  [805] = {x=8.913773, y=-27.596676, z=96.640035, rx=178.000889, ry=-0.000182, rz=-0.000291, shoulder=lefty, elbow=epositive, wrist=wpositive, fatherId=frmaster[2]}
  [806] = {x=7.923867, y=-27.612388, z=96.649585, rx=177.998895, ry=0.000218, rz=-0.000016, shoulder=lefty, elbow=epositive, wrist=wpositive, fatherId=frmaster[2]}
  [807] = {x=6.93352, y=-27.623246, z=96.64007, rx=178.000793, ry=-0.000277, rz=-0.000734, shoulder=lefty, elbow=epositive, wrist=wpositive, fatherId=frmaster[2]}
  [808] = {x=5.944819, y=-27.63732, z=96.640862, rx=178.000734, ry=-0.000326, rz=-0.000446, shoulder=lefty, elbow=epositive, wrist=wpositive, fatherId=frmaster[2]}
  [809] = {x=4.947952, y=-27.654261, z=96.646832, rx=177.999684, ry=-0.000194, rz=-0.000153, shoulder=lefty, elbow=epositive, wrist=wpositive, fatherId=frmaster[2]}
  [810] = {x=3.960147, y=-27.66522, z=96.643162, rx=178.000587, ry=-0.000463, rz=0.000148, shoulder=lefty, elbow=epositive, wrist=wpositive, fatherId=frmaster[2]}
  [811] = {x=2.973867, y=-27.679396, z=96.640369, rx=178.000507, ry=-0.000514, rz=-0.000545, shoulder=lefty, elbow=epositive, wrist=wpositive, fatherId=frmaster[2]}
  [812] = {x=1.979877, y=-27.693391, z=96.637557, rx=178.000612, ry=0.000317, rz=0.000105, shoulder=lefty, elbow=epositive, wrist=wpositive, fatherId=frmaster[2]}
  [813] = {x=0.995231, y=-27.707402, z=96.644933, rx=177.999539, ry=0.000476, rz=-0.000577, shoulder=lefty, elbow=epositive, wrist=wpositive, fatherId=frmaster[2]}
  [814] = {x=0.001401, y=-27.720204, z=96.642841, rx=178.000405, ry=0.000175, rz=-0.000253, shoulder=lefty, elbow=epositive, wrist=wpositive, fatherId=frmaster[2]}
  [815] = {x=-0.983292, y=-27.726863, z=96.644847, rx=178.000296, ry=0.00012, rz=0.000079, shoulder=lefty, elbow=epositive, wrist=wpositive, fatherId=frmaster[2]}
  [816] = {x=-1.976258, y=-27.736283, z=96.642626, rx=178.00017, ry=0.000028, rz=-0.000584, shoulder=lefty, elbow=epositive, wrist=wpositive, fatherId=frmaster[2]}
  [817] = {x=-2.968913, y=-27.743412, z=96.64032, rx=178.000038, ry=-0.000065, rz=-0.000241, shoulder=lefty, elbow=epositive, wrist=wpositive, fatherId=frmaster[2]}
  [818] = {x=-3.960489, y=-27.75152, z=96.648216, rx=177.999898, ry=-0.000158, rz=0.000105, shoulder=lefty, elbow=epositive, wrist=wpositive, fatherId=frmaster[2]}
  [819] = {x=-4.9516, y=-27.758484, z=96.646675, rx=177.999752, ry=-0.000253, rz=0.000459, shoulder=lefty, elbow=epositive, wrist=wpositive, fatherId=frmaster[2]}
  [820] = {x=-5.941493, y=-27.767594, z=96.645991, rx=177.999599, ry=-0.000348, rz=-0.000182, shoulder=lefty, elbow=epositive, wrist=wpositive, fatherId=frmaster[2]}
  [821] = {x=-6.929953, y=-27.77423, z=96.645219, rx=177.999623, ry=0.000476, rz=0.000527, shoulder=lefty, elbow=epositive, wrist=wpositive, fatherId=frmaster[2]}
  [822] = {x=-7.918944, y=-27.78043, z=96.640137, rx=178.000435, ry=0.000184, rz=-0.000102, shoulder=lefty, elbow=epositive, wrist=wpositive, fatherId=frmaster[2]}
  [823] = {x=-8.907014, y=-27.787247, z=96.64016, rx=178.000259, ry=0.000088, rz=0.000274, shoulder=lefty, elbow=epositive, wrist=wpositive, fatherId=frmaster[2]}
  [824] = {x=-9.894404, y=-27.7935, z=96.645241, rx=178.000077, ry=-0.000009, rz=-0.000346, shoulder=lefty, elbow=epositive, wrist=wpositive, fatherId=frmaster[2]}
  [825] = {x=-10.890105, y=-27.802454, z=96.646129, rx=177.999879, ry=-0.000143, rz=0.000038, shoulder=lefty, elbow=epositive, wrist=wpositive, fatherId=frmaster[2]}
  [826] = {x=-11.875867, y=-27.809861, z=96.64268, rx=177.999682, ry=-0.000242, rz=-0.000571, shoulder=lefty, elbow=epositive, wrist=wpositive, fatherId=frmaster[2]}
  [827] = {x=-12.870091, y=-27.818836, z=96.644369, rx=177.99947, ry=-0.000378, rz=-0.000177, shoulder=lefty, elbow=epositive, wrist=wpositive, fatherId=frmaster[2]}
  [828] = {x=-13.853395, y=-27.824988, z=96.651034, rx=177.999433, ry=0.000443, rz=-0.000429, shoulder=lefty, elbow=epositive, wrist=wpositive, fatherId=frmaster[2]}
  [829] = {x=-14.846607, y=-27.832289, z=96.639048, rx=178.000188, ry=0.000122, rz=-0.000021, shoulder=lefty, elbow=epositive, wrist=wpositive, fatherId=frmaster[2]}
  [830] = {x=-15.838709, y=-27.840827, z=96.646606, rx=177.999955, ry=-0.000014, rz=0.000386, shoulder=lefty, elbow=epositive, wrist=wpositive, fatherId=frmaster[2]}
  [831] = {x=-16.830382, y=-27.848304, z=96.64479, rx=177.999714, ry=-0.000152, rz=-0.0002, shoulder=lefty, elbow=epositive, wrist=wpositive, fatherId=frmaster[2]}
  [832] = {x=-17.821399, y=-27.855287, z=96.648035, rx=177.999466, ry=-0.00029, rz=0.000218, shoulder=lefty, elbow=epositive, wrist=wpositive, fatherId=frmaster[2]}
  [833] = {x=-18.810516, y=-27.862721, z=96.647037, rx=177.999375, ry=0.000492, rz=0.000994, shoulder=lefty, elbow=epositive, wrist=wpositive, fatherId=frmaster[2]}
  [834] = {x=-19.800203, y=-27.869818, z=96.641773, rx=178.000097, ry=0.000178, rz=0.000423, shoulder=lefty, elbow=epositive, wrist=wpositive, fatherId=frmaster[2]}
  [835] = {x=-20.789037, y=-27.877666, z=96.641616, rx=177.999827, ry=0.000038, rz=-0.000146, shoulder=lefty, elbow=epositive, wrist=wpositive, fatherId=frmaster[2]}
  [836] = {x=-21.777233, y=-27.885073, z=96.64652, rx=177.999551, ry=-0.000102, rz=0.000288, shoulder=lefty, elbow=epositive, wrist=wpositive, fatherId=frmaster[2]}
  [837] = {x=-22.765223, y=-27.890266, z=96.642039, rx=178.000254, ry=-0.000411, rz=-0.00027, shoulder=lefty, elbow=epositive, wrist=wpositive, fatherId=frmaster[2]}
  [838] = {x=-23.75984, y=-27.900874, z=96.647894, rx=177.999124, ry=0.0005, rz=0.000527, shoulder=lefty, elbow=epositive, wrist=wpositive, fatherId=frmaster[2]}
  [839] = {x=-24.746454, y=-27.906358, z=96.644261, rx=177.999812, ry=0.000193, rz=-0.000023, shoulder=lefty, elbow=epositive, wrist=wpositive, fatherId=frmaster[2]}
  [840] = {x=-25.741373, y=-27.914513, z=96.645809, rx=177.999498, ry=0.000015, rz=0.000428, shoulder=lefty, elbow=epositive, wrist=wpositive, fatherId=frmaster[2]}
  [841] = {x=-26.726631, y=-27.920333, z=96.643032, rx=178.000174, ry=-0.000289, rz=-0.000115, shoulder=lefty, elbow=epositive, wrist=wpositive, fatherId=frmaster[2]}
  [842] = {x=-27.719082, y=-27.928635, z=96.64543, rx=177.999995, ry=0.000455, rz=0.000701, shoulder=lefty, elbow=epositive, wrist=wpositive, fatherId=frmaster[2]}
  [843] = {x=-28.702817, y=-27.936049, z=96.643558, rx=177.999668, ry=0.000311, rz=-0.000835, shoulder=lefty, elbow=epositive, wrist=wpositive, fatherId=frmaster[2]}
  [844] = {x=-29.695588, y=-27.941964, z=96.64167, rx=178.000314, ry=-0.000024, rz=-0.000367, shoulder=lefty, elbow=epositive, wrist=wpositive, fatherId=frmaster[2]}
  [845] = {x=-30.687149, y=-27.951588, z=96.640743, rx=177.999965, ry=-0.000203, rz=0.000102, shoulder=lefty, elbow=epositive, wrist=wpositive, fatherId=frmaster[2]}
  [846] = {x=-31.678617, y=-27.957901, z=96.639728, rx=178.000598, ry=-0.000535, rz=-0.000423, shoulder=lefty, elbow=epositive, wrist=wpositive, fatherId=frmaster[2]}
  [847] = {x=-32.668177, y=-27.964899, z=96.643809, rx=178.000376, ry=0.000208, rz=0.000413, shoulder=lefty, elbow=epositive, wrist=wpositive, fatherId=frmaster[2]}
  [848] = {x=-33.658182, y=-27.972864, z=96.643712, rx=178.000006, ry=0.000028, rz=-0.000106, shoulder=lefty, elbow=epositive, wrist=wpositive, fatherId=frmaster[2]}
  [849] = {x=-34.647604, y=-27.980501, z=96.648675, rx=177.999629, ry=-0.000153, rz=0.000375, shoulder=lefty, elbow=epositive, wrist=wpositive, fatherId=frmaster[2]}
  [850] = {x=-35.636361, y=-27.988956, z=96.64946, rx=177.999245, ry=-0.000335, rz=-0.000139, shoulder=lefty, elbow=epositive, wrist=wpositive, fatherId=frmaster[2]}
  [851] = {x=-36.623808, y=-27.995104, z=96.640917, rx=177.999977, ry=0.000261, rz=-0.000282, shoulder=lefty, elbow=epositive, wrist=wpositive, fatherId=frmaster[2]}
  [852] = {x=-37.620853, y=-28.002846, z=96.646798, rx=177.99957, ry=0.000043, rz=0.000209, shoulder=lefty, elbow=epositive, wrist=wpositive, fatherId=frmaster[2]}
  [853] = {x=-38.608373, y=-28.008476, z=96.639117, rx=178.001145, ry=-0.000417, rz=-0.000292, shoulder=lefty, elbow=epositive, wrist=wpositive, fatherId=frmaster[2]}
  [854] = {x=-39.593779, y=-28.016167, z=96.64585, rx=177.99987, ry=0.000462, rz=-0.000431, shoulder=lefty, elbow=epositive, wrist=wpositive, fatherId=frmaster[2]}
  [855] = {x=-40.58907, y=-28.025203, z=96.639191, rx=178.000432, ry=0.000108, rz=0.000072, shoulder=lefty, elbow=epositive, wrist=wpositive, fatherId=frmaster[2]}
  [856] = {x=-41.574591, y=-28.032435, z=96.646785, rx=178.000006, ry=-0.000073, rz=-0.000427, shoulder=lefty, elbow=epositive, wrist=wpositive, fatherId=frmaster[2]}
  [857] = {x=-42.568912, y=-28.040341, z=96.645196, rx=177.999564, ry=-0.000293, rz=0.000081, shoulder=lefty, elbow=epositive, wrist=wpositive, fatherId=frmaster[2]}
  [858] = {x=-43.552519, y=-28.046198, z=96.63933, rx=178.000236, ry=0.000315, rz=-0.000039, shoulder=lefty, elbow=epositive, wrist=wpositive, fatherId=frmaster[2]}
  [859] = {x=-44.545849, y=-28.053507, z=96.638612, rx=178.000771, ry=-0.000031, rz=-0.000527, shoulder=lefty, elbow=epositive, wrist=wpositive, fatherId=frmaster[2]}
  [860] = {x=-45.538493, y=-28.061772, z=96.642998, rx=178.000309, ry=-0.000249, rz=-0.000015, shoulder=lefty, elbow=epositive, wrist=wpositive, fatherId=frmaster[2]}
  [861] = {x=-46.529424, y=-28.070788, z=96.643232, rx=177.999953, ry=0.000454, rz=0.00087, shoulder=lefty, elbow=epositive, wrist=wpositive, fatherId=frmaster[2]}
  [862] = {x=-47.512248, y=-28.075214, z=96.643319, rx=178.000477, ry=0.000148, rz=-0.00061, shoulder=lefty, elbow=epositive, wrist=wpositive, fatherId=frmaster[2]}
  [863] = {x=-48.503627, y=-28.082047, z=96.639343, rx=178.000985, ry=-0.000191, rz=-0.000086, shoulder=lefty, elbow=epositive, wrist=wpositive, fatherId=frmaster[2]}
  [864] = {x=-49.494351, y=-28.08987, z=96.640474, rx=178.000495, ry=-0.00041, rz=-0.000563, shoulder=lefty, elbow=epositive, wrist=wpositive, fatherId=frmaster[2]}
  [865] = {x=-50.483444, y=-28.097352, z=96.646661, rx=178.000105, ry=0.000294, rz=-0.00067, shoulder=lefty, elbow=epositive, wrist=wpositive, fatherId=frmaster[2]}
  [866] = {x=-51.473202, y=-28.105824, z=96.639482, rx=178.000593, ry=-0.000041, rz=-0.000139, shoulder=lefty, elbow=epositive, wrist=wpositive, fatherId=frmaster[2]}
  [867] = {x=-52.471771, y=-28.113763, z=96.641589, rx=178.000072, ry=-0.000297, rz=0.00039, shoulder=lefty, elbow=epositive, wrist=wpositive, fatherId=frmaster[2]}
  [868] = {x=-53.459292, y=-28.122929, z=96.644577, rx=177.999656, ry=0.000406, rz=0.00029, shoulder=lefty, elbow=epositive, wrist=wpositive, fatherId=frmaster[2]}
  [869] = {x=-54.447712, y=-28.130227, z=96.647541, rx=177.999129, ry=0.000185, rz=-0.000177, shoulder=lefty, elbow=epositive, wrist=wpositive, fatherId=frmaster[2]}
  [870] = {x=-55.435743, y=-28.137278, z=96.646339, rx=177.99959, ry=-0.000144, rz=-0.000641, shoulder=lefty, elbow=epositive, wrist=wpositive, fatherId=frmaster[2]}
  [871] = {x=-56.422416, y=-28.142223, z=96.645109, rx=178.000141, ry=0.000452, rz=-0.000729, shoulder=lefty, elbow=epositive, wrist=wpositive, fatherId=frmaster[2]}
  [872] = {x=-57.41848, y=-28.152621, z=96.644972, rx=177.999584, ry=0.000195, rz=-0.000192, shoulder=lefty, elbow=epositive, wrist=wpositive, fatherId=frmaster[2]}
  [873] = {x=-58.405313, y=-28.158501, z=96.644693, rx=178.000025, ry=-0.000127, rz=-0.000651, shoulder=lefty, elbow=epositive, wrist=wpositive, fatherId=frmaster[2]}
  [874] = {x=-59.400791, y=-28.166654, z=96.640378, rx=178.00045, ry=-0.000484, rz=-0.000107, shoulder=lefty, elbow=epositive, wrist=wpositive, fatherId=frmaster[2]}
  [875] = {x=-60.385354, y=-28.174566, z=96.650304, rx=177.998977, ry=0.000318, rz=-0.000195, shoulder=lefty, elbow=epositive, wrist=wpositive, fatherId=frmaster[2]}
  [876] = {x=-61.380256, y=-28.180496, z=96.641817, rx=178.000384, ry=-0.000133, rz=0.000355, shoulder=lefty, elbow=epositive, wrist=wpositive, fatherId=frmaster[2]}
  [877] = {x=-62.365132, y=-28.18932, z=96.643487, rx=177.999802, ry=-0.000352, rz=-0.000101, shoulder=lefty, elbow=epositive, wrist=wpositive, fatherId=frmaster[2]}
  [878] = {x=-63.357812, y=-28.197297, z=96.64521, rx=177.999289, ry=0.000314, rz=-0.00018, shoulder=lefty, elbow=epositive, wrist=wpositive, fatherId=frmaster[2]}
  [879] = {x=-64.342146, y=-28.203971, z=96.642714, rx=177.999688, ry=0.000002, rz=-0.00063, shoulder=lefty, elbow=epositive, wrist=wpositive, fatherId=frmaster[2]}
  [880] = {x=-65.335411, y=-28.209874, z=96.640279, rx=178.000073, ry=-0.000344, rz=-0.000077, shoulder=lefty, elbow=epositive, wrist=wpositive, fatherId=frmaster[2]}
  [881] = {x=-66.326818, y=-28.218619, z=96.648026, rx=177.999534, ry=0.000325, rz=-0.000157, shoulder=lefty, elbow=epositive, wrist=wpositive, fatherId=frmaster[2]}
  [882] = {x=-67.319242, y=-28.225415, z=96.646555, rx=177.999904, ry=-0.000016, rz=0.000396, shoulder=lefty, elbow=epositive, wrist=wpositive, fatherId=frmaster[2]}
  [883] = {x=-66.317022, y=-28.225289, z=96.64487, rx=177.999542, ry=0.000364, rz=-0.000161, shoulder=lefty, elbow=epositive, wrist=wpositive, fatherId=frmaster[2]}
  [884] = {x=-65.324629, y=-28.226264, z=96.648325, rx=177.999086, ry=-0.000212, rz=-0.000098, shoulder=lefty, elbow=epositive, wrist=wpositive, fatherId=frmaster[2]}
  [885] = {x=-64.321617, y=-28.225732, z=96.647556, rx=177.999707, ry=0.000085, rz=-0.000655, shoulder=lefty, elbow=epositive, wrist=wpositive, fatherId=frmaster[2]}
  [886] = {x=-63.3274, y=-28.225595, z=96.646886, rx=177.999316, ry=0.000435, rz=-0.000209, shoulder=lefty, elbow=epositive, wrist=wpositive, fatherId=frmaster[2]}
  [887] = {x=-62.33406, y=-28.224115, z=96.642027, rx=178.000825, ry=-0.000322, rz=-0.000135, shoulder=lefty, elbow=epositive, wrist=wpositive, fatherId=frmaster[2]}
  [888] = {x=-61.329773, y=-28.223559, z=96.642231, rx=178.000429, ry=0.000066, rz=-0.000688, shoulder=lefty, elbow=epositive, wrist=wpositive, fatherId=frmaster[2]}
  [889] = {x=-60.334157, y=-28.224056, z=96.647574, rx=178.000018, ry=0.000422, rz=-0.000242, shoulder=lefty, elbow=epositive, wrist=wpositive, fatherId=frmaster[2]}
  [890] = {x=-59.339162, y=-28.225622, z=96.648809, rx=177.99951, ry=-0.000143, rz=-0.000168, shoulder=lefty, elbow=epositive, wrist=wpositive, fatherId=frmaster[2]}
  [891] = {x=-58.34288, y=-28.224981, z=96.640795, rx=178.000079, ry=0.000115, rz=0.000289, shoulder=lefty, elbow=epositive, wrist=wpositive, fatherId=frmaster[2]}
  [892] = {x=-57.345756, y=-28.227191, z=96.642969, rx=177.999648, ry=0.000477, rz=0.00074, shoulder=lefty, elbow=epositive, wrist=wpositive, fatherId=frmaster[2]}
  [893] = {x=-56.349631, y=-28.226272, z=96.645077, rx=178.000108, ry=-0.000186, rz=-0.000178, shoulder=lefty, elbow=epositive, wrist=wpositive, fatherId=frmaster[2]}
  [894] = {x=-55.352089, y=-28.224342, z=96.637971, rx=178.000657, ry=0.00007, rz=0.000284, shoulder=lefty, elbow=epositive, wrist=wpositive, fatherId=frmaster[2]}
  [895] = {x=-54.353676, y=-28.225231, z=96.641054, rx=178.000205, ry=0.000437, rz=0.000741, shoulder=lefty, elbow=epositive, wrist=wpositive, fatherId=frmaster[2]}
  [896] = {x=-53.355882, y=-28.226014, z=96.649205, rx=177.999645, ry=-0.000116, rz=-0.000174, shoulder=lefty, elbow=epositive, wrist=wpositive, fatherId=frmaster[2]}
  [897] = {x=-52.35665, y=-28.225759, z=96.648132, rx=177.999178, ry=0.000254, rz=0.00029, shoulder=lefty, elbow=epositive, wrist=wpositive, fatherId=frmaster[2]}
  [898] = {x=-51.357127, y=-28.22397, z=96.64284, rx=178.000693, ry=0.0004, rz=-0.000242, shoulder=lefty, elbow=epositive, wrist=wpositive, fatherId=frmaster[2]}
  [899] = {x=-50.367069, y=-28.22592, z=96.642773, rx=178.000098, ry=-0.000187, rz=0.000855, shoulder=lefty, elbow=epositive, wrist=wpositive, fatherId=frmaster[2]}
  [900] = {x=-49.366217, y=-28.226061, z=96.647685, rx=177.999611, ry=0.00019, rz=0.000322, shoulder=lefty, elbow=epositive, wrist=wpositive, fatherId=frmaster[2]}
  [901] = {x=-48.365182, y=-28.224052, z=96.64332, rx=178.000111, ry=0.000447, rz=-0.000203, shoulder=lefty, elbow=epositive, wrist=wpositive, fatherId=frmaster[2]}
  [902] = {x=-47.373462, y=-28.226399, z=96.649234, rx=177.999491, ry=-0.000132, rz=-0.000102, shoulder=lefty, elbow=epositive, wrist=wpositive, fatherId=frmaster[2]}
  [903] = {x=-46.371288, y=-28.224977, z=96.645782, rx=177.999976, ry=0.000126, rz=-0.000623, shoulder=lefty, elbow=epositive, wrist=wpositive, fatherId=frmaster[2]}
  [904] = {x=-45.377551, y=-28.22599, z=96.647509, rx=177.999453, ry=0.000472, rz=0.000855, shoulder=lefty, elbow=epositive, wrist=wpositive, fatherId=frmaster[2]}
  [905] = {x=-44.375338, y=-28.225258, z=96.644969, rx=177.999807, ry=-0.000192, rz=-0.000029, shoulder=lefty, elbow=epositive, wrist=wpositive, fatherId=frmaster[2]}
  [906] = {x=-43.380854, y=-28.223836, z=96.642461, rx=178.000262, ry=0.000028, rz=-0.000542, shoulder=lefty, elbow=epositive, wrist=wpositive, fatherId=frmaster[2]}
  [907] = {x=-42.385459, y=-28.225042, z=96.640892, rx=178.000711, ry=0.000248, rz=-0.000055, shoulder=lefty, elbow=epositive, wrist=wpositive, fatherId=frmaster[2]}
  [908] = {x=-41.390904, y=-28.224314, z=96.639287, rx=178.001029, ry=-0.000457, rz=0.00007, shoulder=lefty, elbow=epositive, wrist=wpositive, fatherId=frmaster[2]}
  [909] = {x=-40.394487, y=-28.224336, z=96.64278, rx=178.000471, ry=-0.000104, rz=0.000562, shoulder=lefty, elbow=epositive, wrist=wpositive, fatherId=frmaster[2]}
  [910] = {x=-39.388444, y=-28.222336, z=96.641987, rx=178.000907, ry=0.000151, rz=0.000059, shoulder=lefty, elbow=epositive, wrist=wpositive, fatherId=frmaster[2]}
  [911] = {x=-38.391912, y=-28.222977, z=96.64638, rx=178.000208, ry=-0.000415, rz=-0.000808, shoulder=lefty, elbow=epositive, wrist=wpositive, fatherId=frmaster[2]}
  [912] = {x=-37.402718, y=-28.225912, z=96.646671, rx=177.999621, ry=-0.000093, rz=0.000693, shoulder=lefty, elbow=epositive, wrist=wpositive, fatherId=frmaster[2]}
  [913] = {x=-36.403877, y=-28.226772, z=96.642665, rx=178.000027, ry=0.000126, rz=0.000199, shoulder=lefty, elbow=epositive, wrist=wpositive, fatherId=frmaster[2]}
  [914] = {x=-35.404647, y=-28.22558, z=96.647894, rx=177.999437, ry=0.000489, rz=0.000706, shoulder=lefty, elbow=epositive, wrist=wpositive, fatherId=frmaster[2]}
  [915] = {x=-34.406123, y=-28.224032, z=96.639617, rx=178.000682, ry=-0.000361, rz=-0.00014, shoulder=lefty, elbow=epositive, wrist=wpositive, fatherId=frmaster[2]}
  [916] = {x=-33.405599, y=-28.223217, z=96.645724, rx=178.000077, ry=0.000003, rz=-0.000627, shoulder=lefty, elbow=epositive, wrist=wpositive, fatherId=frmaster[2]}
  [917] = {x=-32.413596, y=-28.224812, z=96.638426, rx=178.000446, ry=0.000183, rz=-0.000106, shoulder=lefty, elbow=epositive, wrist=wpositive, fatherId=frmaster[2]}
  [918] = {x=-31.412876, y=-28.224513, z=96.645411, rx=177.999687, ry=-0.000371, rz=0.000054, shoulder=lefty, elbow=epositive, wrist=wpositive, fatherId=frmaster[2]}
  [919] = {x=-30.419445, y=-28.226537, z=96.648273, rx=177.999053, ry=-0.000037, rz=0.000578, shoulder=lefty, elbow=epositive, wrist=wpositive, fatherId=frmaster[2]}
  [920] = {x=-29.416847, y=-28.223345, z=96.64166, rx=178.000396, ry=0.000025, rz=0.000111, shoulder=lefty, elbow=epositive, wrist=wpositive, fatherId=frmaster[2]}
  [921] = {x=-28.422057, y=-28.225676, z=96.64538, rx=177.999749, ry=0.000361, rz=-0.000358, shoulder=lefty, elbow=epositive, wrist=wpositive, fatherId=frmaster[2]}
  [922] = {x=-27.428363, y=-28.224754, z=96.639699, rx=178.000922, ry=-0.000541, rz=-0.000177, shoulder=lefty, elbow=epositive, wrist=wpositive, fatherId=frmaster[2]}
  [923] = {x=-26.432518, y=-28.225634, z=96.639153, rx=178.00026, ry=-0.000204, rz=0.000364, shoulder=lefty, elbow=epositive, wrist=wpositive, fatherId=frmaster[2]}
  [924] = {x=-25.42709, y=-28.222996, z=96.643548, rx=178.000587, ry=0.00001, rz=-0.000091, shoulder=lefty, elbow=epositive, wrist=wpositive, fatherId=frmaster[2]}
  [925] = {x=-24.429846, y=-28.22409, z=96.643847, rx=177.999912, ry=0.000351, rz=-0.000542, shoulder=lefty, elbow=epositive, wrist=wpositive, fatherId=frmaster[2]}
  [926] = {x=-23.433165, y=-28.224831, z=96.639887, rx=178.000062, ry=-0.000394, rz=-0.000344, shoulder=lefty, elbow=epositive, wrist=wpositive, fatherId=frmaster[2]}
  [927] = {x=-22.434701, y=-28.224901, z=96.640978, rx=178.000359, ry=-0.000218, rz=-0.000787, shoulder=lefty, elbow=epositive, wrist=wpositive, fatherId=frmaster[2]}
  [928] = {x=-21.445055, y=-28.224708, z=96.642082, rx=178.00064, ry=-0.000079, rz=0.000775, shoulder=lefty, elbow=epositive, wrist=wpositive, fatherId=frmaster[2]}
  [929] = {x=-20.444948, y=-28.226127, z=96.644044, rx=177.999938, ry=0.000268, rz=0.00034, shoulder=lefty, elbow=epositive, wrist=wpositive, fatherId=frmaster[2]}
  [930] = {x=-19.444725, y=-28.224121, z=96.645899, rx=178.000215, ry=0.000443, rz=-0.00009, shoulder=lefty, elbow=epositive, wrist=wpositive, fatherId=frmaster[2]}
  [931] = {x=-18.453978, y=-28.224908, z=96.643598, rx=178.000312, ry=-0.000341, rz=0.000134, shoulder=lefty, elbow=epositive, wrist=wpositive, fatherId=frmaster[2]}
  [932] = {x=-17.452082, y=-28.22418, z=96.646314, rx=177.999589, ry=0.000009, rz=-0.000286, shoulder=lefty, elbow=epositive, wrist=wpositive, fatherId=frmaster[2]}
  [933] = {x=-16.458737, y=-28.224849, z=96.644818, rx=177.999835, ry=0.000147, rz=0.000298, shoulder=lefty, elbow=epositive, wrist=wpositive, fatherId=frmaster[2]}
  [934] = {x=-15.45567, y=-28.222866, z=96.638949, rx=178.001066, ry=0.000138, rz=-0.000111, shoulder=lefty, elbow=epositive, wrist=wpositive, fatherId=frmaster[2]}
  [935] = {x=-14.461962, y=-28.223766, z=96.63826, rx=178.001126, ry=-0.000649, rz=0.000133, shoulder=lefty, elbow=epositive, wrist=wpositive, fatherId=frmaster[2]}
  [936] = {x=-13.466218, y=-28.225093, z=96.642665, rx=178.000367, ry=-0.000331, rz=-0.000269, shoulder=lefty, elbow=epositive, wrist=wpositive, fatherId=frmaster[2]}
  [937] = {x=-12.469648, y=-28.226968, z=96.642808, rx=177.999601, ry=-0.000011, rz=0.000335, shoulder=lefty, elbow=epositive, wrist=wpositive, fatherId=frmaster[2]}
  [938] = {x=-11.473203, y=-28.224185, z=96.642789, rx=178.000793, ry=-0.000065, rz=0.000944, shoulder=lefty, elbow=epositive, wrist=wpositive, fatherId=frmaster[2]}
  [939] = {x=-10.475105, y=-28.225985, z=96.64372, rx=178.000014, ry=0.000257, rz=0.000558, shoulder=lefty, elbow=epositive, wrist=wpositive, fatherId=frmaster[2]}
  [940] = {x=-9.476304, y=-28.227157, z=96.649709, rx=177.999229, ry=0.000582, rz=0.000176, shoulder=lefty, elbow=epositive, wrist=wpositive, fatherId=frmaster[2]}
  [941] = {x=-8.478387, y=-28.226192, z=96.646247, rx=177.999237, ry=-0.000205, rz=0.000456, shoulder=lefty, elbow=epositive, wrist=wpositive, fatherId=frmaster[2]}
  [942] = {x=-7.478737, y=-28.22429, z=96.638447, rx=178.000399, ry=-0.000269, rz=0.000088, shoulder=lefty, elbow=epositive, wrist=wpositive, fatherId=frmaster[2]}
  [943] = {x=-6.477678, y=-28.22463, z=96.650274, rx=177.999592, ry=0.000059, rz=-0.000278, shoulder=lefty, elbow=epositive, wrist=wpositive, fatherId=frmaster[2]}
  [944] = {x=-5.485365, y=-28.225923, z=96.643354, rx=177.99975, ry=0.000153, rz=0.000364, shoulder=lefty, elbow=epositive, wrist=wpositive, fatherId=frmaster[2]}
  [945] = {x=-4.483205, y=-28.224322, z=96.641409, rx=177.99991, ry=0.000283, rz=0.000011, shoulder=lefty, elbow=epositive, wrist=wpositive, fatherId=frmaster[2]}
  [946] = {x=-3.48947, y=-28.224263, z=96.644598, rx=178.000055, ry=0.000375, rz=-0.000337, shoulder=lefty, elbow=epositive, wrist=wpositive, fatherId=frmaster[2]}
  [947] = {x=-2.495993, y=-28.224874, z=96.64349, rx=178, ry=-0.000454, rz=-0.000019, shoulder=lefty, elbow=epositive, wrist=wpositive, fatherId=frmaster[2]}
  [948] = {x=-1.500768, y=-28.224476, z=96.63802, rx=178.001107, ry=-0.000569, rz=0.000646, shoulder=lefty, elbow=epositive, wrist=wpositive, fatherId=frmaster[2]}
  [949] = {x=-0.494798, y=-28.22505, z=96.64276, rx=178.000259, ry=-0.000237, rz=-0.000683, shoulder=lefty, elbow=epositive, wrist=wpositive, fatherId=frmaster[2]}
  [950] = {x=0.502375, y=-28.225555, z=96.647483, rx=177.999395, ry=0.000062, rz=-0.000007, shoulder=lefty, elbow=epositive, wrist=wpositive, fatherId=frmaster[2]}
  [951] = {x=1.500179, y=-28.225235, z=96.647844, rx=177.999503, ry=0.000152, rz=-0.000325, shoulder=lefty, elbow=epositive, wrist=wpositive, fatherId=frmaster[2]}
  [952] = {x=2.489735, y=-28.227623, z=96.64395, rx=177.999595, ry=0.000204, rz=0.000364, shoulder=lefty, elbow=epositive, wrist=wpositive, fatherId=frmaster[2]}
  [953] = {x=3.489154, y=-28.226882, z=96.645034, rx=177.999689, ry=0.000292, rz=0.000059, shoulder=lefty, elbow=epositive, wrist=wpositive, fatherId=frmaster[2]}
  [954] = {x=4.489471, y=-28.226459, z=96.641778, rx=177.999776, ry=0.000379, rz=-0.000239, shoulder=lefty, elbow=epositive, wrist=wpositive, fatherId=frmaster[2]}
  [955] = {x=5.480714, y=-28.224849, z=96.63845, rx=178.000822, ry=0.00021, rz=0.000468, shoulder=lefty, elbow=epositive, wrist=wpositive, fatherId=frmaster[2]}
  [956] = {x=6.48163, y=-28.22423, z=96.645354, rx=177.999711, ry=-0.000406, rz=-0.00015, shoulder=lefty, elbow=epositive, wrist=wpositive, fatherId=frmaster[2]}
  [957] = {x=7.475075, y=-28.224809, z=96.638485, rx=178.000741, ry=-0.00058, rz=0.000572, shoulder=lefty, elbow=epositive, wrist=wpositive, fatherId=frmaster[2]}
  [958] = {x=8.478756, y=-28.223343, z=96.646085, rx=177.999822, ry=-0.000275, rz=-0.000699, shoulder=lefty, elbow=epositive, wrist=wpositive, fatherId=frmaster[2]}
  [959] = {x=9.474525, y=-28.226077, z=96.64511, rx=177.999863, ry=-0.000228, rz=0.000036, shoulder=lefty, elbow=epositive, wrist=wpositive, fatherId=frmaster[2]}
  [960] = {x=10.470626, y=-28.22637, z=96.64402, rx=177.999897, ry=-0.000183, rz=-0.000222, shoulder=lefty, elbow=epositive, wrist=wpositive, fatherId=frmaster[2]}
  [961] = {x=11.467741, y=-28.226958, z=96.648024, rx=177.99895, ry=0.000091, rz=0.000527, shoulder=lefty, elbow=epositive, wrist=wpositive, fatherId=frmaster[2]}
  [962] = {x=12.465216, y=-28.225379, z=96.64757, rx=177.999942, ry=-0.000095, rz=0.000284, shoulder=lefty, elbow=epositive, wrist=wpositive, fatherId=frmaster[2]}
  [963] = {x=13.463895, y=-28.22518, z=96.642775, rx=177.999954, ry=-0.000052, rz=0.000048, shoulder=lefty, elbow=epositive, wrist=wpositive, fatherId=frmaster[2]}
  [964] = {x=14.463311, y=-28.224033, z=96.643028, rx=177.999959, ry=-0.000011, rz=-0.000181, shoulder=lefty, elbow=epositive, wrist=wpositive, fatherId=frmaster[2]}
  [965] = {x=15.454229, y=-28.224436, z=96.638922, rx=178.000919, ry=-0.000242, rz=0.000596, shoulder=lefty, elbow=epositive, wrist=wpositive, fatherId=frmaster[2]}
  [966] = {x=16.456014, y=-28.225182, z=96.645047, rx=177.999938, ry=0.000034, rz=0.000383, shoulder=lefty, elbow=epositive, wrist=wpositive, fatherId=frmaster[2]}
  [967] = {x=17.44889, y=-28.22595, z=96.64163, rx=177.999912, ry=0.000037, rz=0.000176, shoulder=lefty, elbow=epositive, wrist=wpositive, fatherId=frmaster[2]}
  [968] = {x=18.452056, y=-28.224603, z=96.648365, rx=177.999888, ry=0.000076, rz=-0.000022, shoulder=lefty, elbow=epositive, wrist=wpositive, fatherId=frmaster[2]}
  [969] = {x=19.446603, y=-28.224474, z=96.645585, rx=177.999848, ry=0.000077, rz=-0.000214, shoulder=lefty, elbow=epositive, wrist=wpositive, fatherId=frmaster[2]}
  [970] = {x=20.442509, y=-28.225935, z=96.643567, rx=177.999801, ry=0.000077, rz=0.000603, shoulder=lefty, elbow=epositive, wrist=wpositive, fatherId=frmaster[2]}
  [971] = {x=21.439152, y=-28.226339, z=96.646595, rx=177.999746, ry=0.000077, rz=0.000428, shoulder=lefty, elbow=epositive, wrist=wpositive, fatherId=frmaster[2]}
  [972] = {x=22.436737, y=-28.226786, z=96.645194, rx=177.999684, ry=0.000076, rz=0.000261, shoulder=lefty, elbow=epositive, wrist=wpositive, fatherId=frmaster[2]}
  [973] = {x=23.435055, y=-28.226138, z=96.648841, rx=177.999615, ry=0.000074, rz=0.000103, shoulder=lefty, elbow=epositive, wrist=wpositive, fatherId=frmaster[2]}
  [974] = {x=24.434317, y=-28.225493, z=96.648049, rx=177.999538, ry=0.000071, rz=-0.000047, shoulder=lefty, elbow=epositive, wrist=wpositive, fatherId=frmaster[2]}
  [975] = {x=25.434214, y=-28.22365, z=96.642768, rx=178.000421, ry=-0.000187, rz=-0.000189, shoulder=lefty, elbow=epositive, wrist=wpositive, fatherId=frmaster[2]}
  [976] = {x=26.426013, y=-28.224608, z=96.642646, rx=178.000321, ry=-0.000229, rz=-0.000323, shoulder=lefty, elbow=epositive, wrist=wpositive, fatherId=frmaster[2]}
  [977] = {x=27.428324, y=-28.224206, z=96.643183, rx=178.000222, ry=-0.000236, rz=-0.000447, shoulder=lefty, elbow=epositive, wrist=wpositive, fatherId=frmaster[2]}
  [978] = {x=28.422544, y=-28.226585, z=96.648882, rx=177.999141, ry=-0.000021, rz=-0.000562, shoulder=lefty, elbow=epositive, wrist=wpositive, fatherId=frmaster[2]}
  [979] = {x=29.416646, y=-28.225088, z=96.644837, rx=177.999984, ry=-0.000325, rz=0.00033, shoulder=lefty, elbow=epositive, wrist=wpositive, fatherId=frmaster[2]}
  [980] = {x=30.412443, y=-28.226121, z=96.641553, rx=177.999854, ry=-0.000371, rz=0.000232, shoulder=lefty, elbow=epositive, wrist=wpositive, fatherId=frmaster[2]}
  [981] = {x=31.418857, y=-28.225665, z=96.648475, rx=177.998761, ry=-0.000117, rz=-0.000854, shoulder=lefty, elbow=epositive, wrist=wpositive, fatherId=frmaster[2]}
  [982] = {x=32.407986, y=-28.226693, z=96.64577, rx=177.999825, ry=0.000453, rz=0.000372, shoulder=lefty, elbow=epositive, wrist=wpositive, fatherId=frmaster[2]}
  [983] = {x=33.406073, y=-28.225007, z=96.638504, rx=178.000638, ry=0.000137, rz=0.0003, shoulder=lefty, elbow=epositive, wrist=wpositive, fatherId=frmaster[2]}
  [984] = {x=34.405638, y=-28.224612, z=96.64152, rx=178.000479, ry=0.000087, rz=0.00024, shoulder=lefty, elbow=epositive, wrist=wpositive, fatherId=frmaster[2]}
  [985] = {x=35.406149, y=-28.224001, z=96.640033, rx=178.000313, ry=0.000036, rz=0.000188, shoulder=lefty, elbow=epositive, wrist=wpositive, fatherId=frmaster[2]}
  [986] = {x=36.398234, y=-28.224987, z=96.643659, rx=178.000131, ry=-0.000053, rz=0.000146, shoulder=lefty, elbow=epositive, wrist=wpositive, fatherId=frmaster[2]}
  [987] = {x=37.400836, y=-28.224171, z=96.647906, rx=177.99995, ry=-0.000106, rz=0.000115, shoulder=lefty, elbow=epositive, wrist=wpositive, fatherId=frmaster[2]}
  [988] = {x=38.394468, y=-28.223487, z=96.642454, rx=178.000714, ry=-0.000471, rz=0.000092, shoulder=lefty, elbow=epositive, wrist=wpositive, fatherId=frmaster[2]}
  [989] = {x=39.389818, y=-28.225083, z=96.637721, rx=178.000509, ry=-0.000563, rz=0.000079, shoulder=lefty, elbow=epositive, wrist=wpositive, fatherId=frmaster[2]}
  [990] = {x=40.387769, y=-28.227479, z=96.643265, rx=177.999603, ry=0.00054, rz=0.000377, shoulder=lefty, elbow=epositive, wrist=wpositive, fatherId=frmaster[2]}
  [991] = {x=41.384414, y=-28.22615, z=96.63898, rx=178.000345, ry=0.000167, rz=0.000384, shoulder=lefty, elbow=epositive, wrist=wpositive, fatherId=frmaster[2]}
  [992] = {x=42.382531, y=-28.225889, z=96.644988, rx=178.000119, ry=0.000073, rz=0.000404, shoulder=lefty, elbow=epositive, wrist=wpositive, fatherId=frmaster[2]}
  [993] = {x=43.381582, y=-28.225241, z=96.646444, rx=177.999885, ry=-0.000022, rz=0.000433, shoulder=lefty, elbow=epositive, wrist=wpositive, fatherId=frmaster[2]}
  [994] = {x=44.381214, y=-28.223014, z=96.643298, rx=178.000602, ry=-0.000404, rz=-0.000528, shoulder=lefty, elbow=epositive, wrist=wpositive, fatherId=frmaster[2]}
  [995] = {x=45.373431, y=-28.225964, z=96.64092, rx=178.000344, ry=-0.000538, rz=0.000522, shoulder=lefty, elbow=epositive, wrist=wpositive, fatherId=frmaster[2]}
  [996] = {x=46.376576, y=-28.223909, z=96.643482, rx=178.000364, ry=0.000279, rz=-0.000124, shoulder=lefty, elbow=epositive, wrist=wpositive, fatherId=frmaster[2]}
  [997] = {x=47.370389, y=-28.224837, z=96.64155, rx=178.000093, ry=0.000143, rz=-0.000053, shoulder=lefty, elbow=epositive, wrist=wpositive, fatherId=frmaster[2]}
  [998] = {x=48.365209, y=-28.225428, z=96.640215, rx=178.00077, ry=-0.000286, rz=0.00003, shoulder=lefty, elbow=epositive, wrist=wpositive, fatherId=frmaster[2]}
  [999] = {x=49.361041, y=-28.225561, z=96.643946, rx=178.000482, ry=-0.000425, rz=0.000126, shoulder=lefty, elbow=epositive, wrist=wpositive, fatherId=frmaster[2]}
  [1000] = {x=50.358593, y=-28.227613, z=96.648352, rx=177.999232, ry=-0.000268, rz=0.000235, shoulder=lefty, elbow=epositive, wrist=wpositive, fatherId=frmaster[2]}
  [1001] = {x=51.357811, y=-28.227567, z=96.648097, rx=177.999216, ry=0.000509, rz=0.000638, shoulder=lefty, elbow=epositive, wrist=wpositive, fatherId=frmaster[2]}
  [1002] = {x=52.356451, y=-28.226097, z=96.643194, rx=177.999862, ry=0.000071, rz=-0.000234, shoulder=lefty, elbow=epositive, wrist=wpositive, fatherId=frmaster[2]}
  [1003] = {x=53.356534, y=-28.22533, z=96.648589, rx=177.999546, ry=-0.000071, rz=-0.00009, shoulder=lefty, elbow=epositive, wrist=wpositive, fatherId=frmaster[2]}
  [1004] = {x=54.348375, y=-28.227155, z=96.649431, rx=177.999213, ry=-0.000248, rz=0.000063, shoulder=lefty, elbow=epositive, wrist=wpositive, fatherId=frmaster[2]}
  [1005] = {x=55.350989, y=-28.22352, z=96.645506, rx=178.000127, ry=0.00022, rz=-0.000493, shoulder=lefty, elbow=epositive, wrist=wpositive, fatherId=frmaster[2]}
  [1006] = {x=56.344676, y=-28.22407, z=96.642263, rx=178.000731, ry=-0.000267, rz=-0.000316, shoulder=lefty, elbow=epositive, wrist=wpositive, fatherId=frmaster[2]}
  [1007] = {x=57.340064, y=-28.226303, z=96.639647, rx=178.000376, ry=-0.00045, rz=-0.000126, shoulder=lefty, elbow=epositive, wrist=wpositive, fatherId=frmaster[2]}
  [1008] = {x=58.337166, y=-28.226302, z=96.64203, rx=178.000311, ry=0.00028, rz=0.000353, shoulder=lefty, elbow=epositive, wrist=wpositive, fatherId=frmaster[2]}
  [1009] = {x=59.334464, y=-28.227101, z=96.645008, rx=177.999942, ry=0.000096, rz=0.00057, shoulder=lefty, elbow=epositive, wrist=wpositive, fatherId=frmaster[2]}
  [1010] = {x=60.332624, y=-28.227067, z=96.64331, rx=177.999565, ry=-0.000088, rz=-0.000202, shoulder=lefty, elbow=epositive, wrist=wpositive, fatherId=frmaster[2]}
  [1011] = {x=61.332818, y=-28.225859, z=96.642126, rx=178.000433, ry=0.000325, rz=0.000312, shoulder=lefty, elbow=epositive, wrist=wpositive, fatherId=frmaster[2]}
  [1012] = {x=62.332841, y=-28.224177, z=96.646001, rx=178.000041, ry=0.000138, rz=-0.000432, shoulder=lefty, elbow=epositive, wrist=wpositive, fatherId=frmaster[2]}
  [1013] = {x=63.324912, y=-28.226127, z=96.640764, rx=178.000582, ry=-0.000404, rz=-0.000166, shoulder=lefty, elbow=epositive, wrist=wpositive, fatherId=frmaster[2]}
  [1014] = {x=64.328168, y=-28.223389, z=96.640477, rx=178.000482, ry=0.00032, rz=-0.000617, shoulder=lefty, elbow=epositive, wrist=wpositive, fatherId=frmaster[2]}
  [1015] = {x=65.322441, y=-28.224665, z=96.640823, rx=178.00006, ry=0.000093, rz=-0.000322, shoulder=lefty, elbow=epositive, wrist=wpositive, fatherId=frmaster[2]}
  [1016] = {x=66.31758, y=-28.224954, z=96.641667, rx=178.000576, ry=-0.000457, rz=-0.000011, shoulder=lefty, elbow=epositive, wrist=wpositive, fatherId=frmaster[2]}
  [1017] = {x=67.315477, y=-28.226134, z=96.64307, rx=178.000451, ry=0.000226, rz=0.000577, shoulder=lefty, elbow=epositive, wrist=wpositive, fatherId=frmaster[2]}
  [1018] = {x=66.314886, y=-28.216949, z=96.64457, rx=177.999631, ry=-0.000133, rz=-0.000018, shoulder=lefty, elbow=epositive, wrist=wpositive, fatherId=frmaster[2]}
  [1019] = {x=65.325405, y=-28.202804, z=96.646455, rx=178.00007, ry=0.000133, rz=-0.000334, shoulder=lefty, elbow=epositive, wrist=wpositive, fatherId=frmaster[2]}
  [1020] = {x=64.327612, y=-28.191022, z=96.643675, rx=178.000493, ry=0.000362, rz=-0.000639, shoulder=lefty, elbow=epositive, wrist=wpositive, fatherId=frmaster[2]}
  [1021] = {x=63.330809, y=-28.18209, z=96.646737, rx=177.999654, ry=-0.000006, rz=-0.000194, shoulder=lefty, elbow=epositive, wrist=wpositive, fatherId=frmaster[2]}
  [1022] = {x=62.326436, y=-28.174007, z=96.645098, rx=178.000053, ry=0.000184, rz=0.00053, shoulder=lefty, elbow=epositive, wrist=wpositive, fatherId=frmaster[2]}
  [1023] = {x=61.330931, y=-28.161885, z=96.638688, rx=178.000151, ry=-0.000504, rz=-0.000005, shoulder=lefty, elbow=epositive, wrist=wpositive, fatherId=frmaster[2]}
  [1024] = {x=60.337557, y=-28.148547, z=96.642509, rx=178.000545, ry=-0.000279, rz=-0.000252, shoulder=lefty, elbow=epositive, wrist=wpositive, fatherId=frmaster[2]}
  [1025] = {x=59.33674, y=-28.140028, z=96.646993, rx=177.999973, ry=0.00022, rz=0.000515, shoulder=lefty, elbow=epositive, wrist=wpositive, fatherId=frmaster[2]}
  [1026] = {x=58.345155, y=-28.128809, z=96.642255, rx=178.000053, ry=-0.000472, rz=-0.000981, shoulder=lefty, elbow=epositive, wrist=wpositive, fatherId=frmaster[2]}
  [1027] = {x=57.346527, y=-28.11976, z=96.642617, rx=177.999465, ry=0.000021, rz=-0.00019, shoulder=lefty, elbow=epositive, wrist=wpositive, fatherId=frmaster[2]}
  [1028] = {x=56.348129, y=-28.107602, z=96.647932, rx=177.99982, ry=0.000203, rz=-0.000384, shoulder=lefty, elbow=epositive, wrist=wpositive, fatherId=frmaster[2]}
  [1029] = {x=55.351346, y=-28.09699, z=96.64416, rx=178.000168, ry=0.000385, rz=-0.000567, shoulder=lefty, elbow=epositive, wrist=wpositive, fatherId=frmaster[2]}
  [1030] = {x=54.354069, y=-28.084851, z=96.6454, rx=178.000216, ry=-0.000348, rz=-0.000017, shoulder=lefty, elbow=epositive, wrist=wpositive, fatherId=frmaster[2]}
  [1031] = {x=53.350396, y=-28.077228, z=96.637645, rx=178.000541, ry=-0.000203, rz=0.000823, shoulder=lefty, elbow=epositive, wrist=wpositive, fatherId=frmaster[2]}
  [1032] = {x=52.357405, y=-28.067039, z=96.649782, rx=177.998959, ry=0.000576, rz=-0.000318, shoulder=lefty, elbow=epositive, wrist=wpositive, fatherId=frmaster[2]}
  [1033] = {x=51.363742, y=-28.055304, z=96.647569, rx=177.99899, ry=-0.000163, rz=-0.000735, shoulder=lefty, elbow=epositive, wrist=wpositive, fatherId=frmaster[2]}
  [1034] = {x=50.36262, y=-28.044597, z=96.640756, rx=178.000248, ry=-0.00032, rz=0.000141, shoulder=lefty, elbow=epositive, wrist=wpositive, fatherId=frmaster[2]}
  [1035] = {x=49.363327, y=-28.03577, z=96.644266, rx=177.999587, ry=0.000115, rz=0.000033, shoulder=lefty, elbow=epositive, wrist=wpositive, fatherId=frmaster[2]}
  [1036] = {x=48.364601, y=-28.025159, z=96.643122, rx=177.999874, ry=0.000253, rz=0.000935, shoulder=lefty, elbow=epositive, wrist=wpositive, fatherId=frmaster[2]}
  [1037] = {x=47.367252, y=-28.01528, z=96.642601, rx=178.000154, ry=0.000389, rz=0.000851, shoulder=lefty, elbow=epositive, wrist=wpositive, fatherId=frmaster[2]}
  [1038] = {x=46.369018, y=-28.002747, z=96.641877, rx=178.000148, ry=-0.00039, rz=0.000485, shoulder=lefty, elbow=epositive, wrist=wpositive, fatherId=frmaster[2]}
  [1039] = {x=45.374087, y=-27.993177, z=96.647037, rx=177.999456, ry=0.000033, rz=0.000423, shoulder=lefty, elbow=epositive, wrist=wpositive, fatherId=frmaster[2]}
  [1040] = {x=44.37895, y=-27.979431, z=96.642308, rx=178.000672, ry=-0.00012, rz=0.00037, shoulder=lefty, elbow=epositive, wrist=wpositive, fatherId=frmaster[2]}
  [1041] = {x=43.385555, y=-27.967727, z=96.638268, rx=178.000922, ry=0.000014, rz=-0.000671, shoulder=lefty, elbow=epositive, wrist=wpositive, fatherId=frmaster[2]}
  [1042] = {x=42.384518, y=-27.960056, z=96.644579, rx=178.000197, ry=0.000393, rz=0.000302, shoulder=lefty, elbow=epositive, wrist=wpositive, fatherId=frmaster[2]}
  [1043] = {x=41.382524, y=-27.949734, z=96.641077, rx=178.000154, ry=-0.000428, rz=-0.000016, shoulder=lefty, elbow=epositive, wrist=wpositive, fatherId=frmaster[2]}
  [1044] = {x=40.392179, y=-27.937008, z=96.63815, rx=178.000383, ry=-0.000298, rz=-0.000024, shoulder=lefty, elbow=epositive, wrist=wpositive, fatherId=frmaster[2]}
  [1045] = {x=39.394198, y=-27.928368, z=96.645572, rx=177.999635, ry=0.000072, rz=-0.00002, shoulder=lefty, elbow=epositive, wrist=wpositive, fatherId=frmaster[2]}
  [1046] = {x=38.396394, y=-27.91681, z=96.643193, rx=177.99984, ry=0.000163, rz=-0.000008, shoulder=lefty, elbow=epositive, wrist=wpositive, fatherId=frmaster[2]}
  [1047] = {x=37.399992, y=-27.906301, z=96.64149, rx=178.000037, ry=0.000252, rz=0.000015, shoulder=lefty, elbow=epositive, wrist=wpositive, fatherId=frmaster[2]}
  [1048] = {x=36.404317, y=-27.894368, z=96.644808, rx=178.000226, ry=0.00034, rz=0.000049, shoulder=lefty, elbow=epositive, wrist=wpositive, fatherId=frmaster[2]}
  [1049] = {x=35.399358, y=-27.885394, z=96.643686, rx=178.000141, ry=-0.000524, rz=-0.000213, shoulder=lefty, elbow=epositive, wrist=wpositive, fatherId=frmaster[2]}
  [1050] = {x=34.406054, y=-27.874304, z=96.643167, rx=178.000317, ry=-0.000438, rz=-0.00016, shoulder=lefty, elbow=epositive, wrist=wpositive, fatherId=frmaster[2]}
  [1051] = {x=33.404684, y=-27.865943, z=96.647787, rx=177.999514, ry=-0.00012, rz=-0.000097, shoulder=lefty, elbow=epositive, wrist=wpositive, fatherId=frmaster[2]}
  [1052] = {x=32.413083, y=-27.853285, z=96.647783, rx=177.999675, ry=-0.000037, rz=-0.000024, shoulder=lefty, elbow=epositive, wrist=wpositive, fatherId=frmaster[2]}
  [1053] = {x=31.413322, y=-27.843302, z=96.643358, rx=177.999819, ry=0.00001, rz=0.000057, shoulder=lefty, elbow=epositive, wrist=wpositive, fatherId=frmaster[2]}
  [1054] = {x=30.415062, y=-27.834626, z=96.649199, rx=177.998992, ry=0.000318, rz=0.000149, shoulder=lefty, elbow=epositive, wrist=wpositive, fatherId=frmaster[2]}
  [1055] = {x=29.416697, y=-27.821982, z=96.645274, rx=178.000086, ry=0.0001, rz=0.000249, shoulder=lefty, elbow=epositive, wrist=wpositive, fatherId=frmaster[2]}
  [1056] = {x=28.420058, y=-27.811815, z=96.642107, rx=178.000209, ry=0.000144, rz=0.00036, shoulder=lefty, elbow=epositive, wrist=wpositive, fatherId=frmaster[2]}
  [1057] = {x=27.424169, y=-27.800412, z=96.643971, rx=178.000323, ry=0.000187, rz=0.00048, shoulder=lefty, elbow=epositive, wrist=wpositive, fatherId=frmaster[2]}
  [1058] = {x=26.429252, y=-27.788909, z=96.641367, rx=178.000431, ry=0.000229, rz=-0.000392, shoulder=lefty, elbow=epositive, wrist=wpositive, fatherId=frmaster[2]}
  [1059] = {x=25.435832, y=-27.778865, z=96.649022, rx=177.999564, ry=0.000524, rz=-0.000253, shoulder=lefty, elbow=epositive, wrist=wpositive, fatherId=frmaster[2]}
  [1060] = {x=24.433513, y=-27.768855, z=96.647064, rx=177.999648, ry=0.000526, rz=-0.000107, shoulder=lefty, elbow=epositive, wrist=wpositive, fatherId=frmaster[2]}
  [1061] = {x=23.432592, y=-27.760261, z=96.645843, rx=177.999724, ry=0.000528, rz=0.001048, shoulder=lefty, elbow=epositive, wrist=wpositive, fatherId=frmaster[2]}
  [1062] = {x=22.440011, y=-27.7466, z=96.644406, rx=177.999565, ry=-0.000353, rz=-0.000108, shoulder=lefty, elbow=epositive, wrist=wpositive, fatherId=frmaster[2]}
  [1063] = {x=21.44082, y=-27.736841, z=96.643779, rx=177.999628, ry=-0.000354, rz=0.000064, shoulder=lefty, elbow=epositive, wrist=wpositive, fatherId=frmaster[2]}
  [1064] = {x=20.442296, y=-27.7259, z=96.63868, rx=178.000654, ry=-0.000601, rz=0.000243, shoulder=lefty, elbow=epositive, wrist=wpositive, fatherId=frmaster[2]}
  [1065] = {x=19.444836, y=-27.715046, z=96.638659, rx=178.000703, ry=-0.000602, rz=0.000431, shoulder=lefty, elbow=epositive, wrist=wpositive, fatherId=frmaster[2]}
  [1066] = {x=18.449154, y=-27.707002, z=96.648929, rx=177.998804, ry=-0.000119, rz=-0.000372, shoulder=lefty, elbow=epositive, wrist=wpositive, fatherId=frmaster[2]}
  [1067] = {x=17.453326, y=-27.695076, z=96.640029, rx=177.999808, ry=-0.000366, rz=-0.000168, shoulder=lefty, elbow=epositive, wrist=wpositive, fatherId=frmaster[2]}
  [1068] = {x=16.458361, y=-27.682178, z=96.645655, rx=177.999835, ry=-0.000371, rz=-0.000956, shoulder=lefty, elbow=epositive, wrist=wpositive, fatherId=frmaster[2]}
  [1069] = {x=15.455846, y=-27.674619, z=96.642681, rx=177.999846, ry=-0.000413, rz=0.000264, shoulder=lefty, elbow=epositive, wrist=wpositive, fatherId=frmaster[2]}
  [1070] = {x=14.462518, y=-27.660747, z=96.639458, rx=178.00083, ry=-0.000656, rz=-0.000508, shoulder=lefty, elbow=epositive, wrist=wpositive, fatherId=frmaster[2]}
  [1071] = {x=13.462943, y=-27.652093, z=96.646589, rx=178.000075, ry=0.000454, rz=0.000055, shoulder=lefty, elbow=epositive, wrist=wpositive, fatherId=frmaster[2]}
  [1072] = {x=12.463198, y=-27.643848, z=96.649336, rx=177.99909, ry=0.00064, rz=0.000299, shoulder=lefty, elbow=epositive, wrist=wpositive, fatherId=frmaster[2]}
  [1073] = {x=11.472554, y=-27.629314, z=96.642375, rx=178.000052, ry=0.000399, rz=-0.000449, shoulder=lefty, elbow=epositive, wrist=wpositive, fatherId=frmaster[2]}
  [1074] = {x=10.474244, y=-27.619104, z=96.645736, rx=178.000025, ry=0.000351, rz=-0.00019, shoulder=lefty, elbow=epositive, wrist=wpositive, fatherId=frmaster[2]}
  [1075] = {x=9.476883, y=-27.609088, z=96.644722, rx=177.99999, ry=0.000303, rz=0.000076, shoulder=lefty, elbow=epositive, wrist=wpositive, fatherId=frmaster[2]}
  [1076] = {x=8.480285, y=-27.598163, z=96.648747, rx=177.999949, ry=0.000254, rz=-0.000651, shoulder=lefty, elbow=epositive, wrist=wpositive, fatherId=frmaster[2]}
  [1077] = {x=7.475507, y=-27.589912, z=96.648482, rx=177.999892, ry=0.000168, rz=0.000629, shoulder=lefty, elbow=epositive, wrist=wpositive, fatherId=frmaster[2]}
  [1078] = {x=6.480794, y=-27.579451, z=96.643786, rx=177.999836, ry=0.000117, rz=-0.000084, shoulder=lefty, elbow=epositive, wrist=wpositive, fatherId=frmaster[2]}
  [1079] = {x=5.486172, y=-27.565353, z=96.638934, rx=178.000749, ry=-0.000155, rz=0.000211, shoulder=lefty, elbow=epositive, wrist=wpositive, fatherId=frmaster[2]}
  [1080] = {x=4.484127, y=-27.556776, z=96.644438, rx=177.999695, ry=-0.000025, rz=0.000511, shoulder=lefty, elbow=epositive, wrist=wpositive, fatherId=frmaster[2]}
  [1081] = {x=3.491871, y=-27.544904, z=96.645477, rx=177.999618, ry=-0.000079, rz=-0.000181, shoulder=lefty, elbow=epositive, wrist=wpositive, fatherId=frmaster[2]}
  [1082] = {x=2.491158, y=-27.534519, z=96.642213, rx=178.000502, ry=-0.000385, rz=0.000133, shoulder=lefty, elbow=epositive, wrist=wpositive, fatherId=frmaster[2]}
  [1083] = {x=1.491466, y=-27.524506, z=96.644033, rx=178.000403, ry=-0.000475, rz=0.000453, shoulder=lefty, elbow=epositive, wrist=wpositive, fatherId=frmaster[2]}
  [1084] = {x=0.502943, y=-27.512253, z=96.64144, rx=178.000503, ry=0.000389, rz=0.000121, shoulder=lefty, elbow=epositive, wrist=wpositive, fatherId=frmaster[2]}
  [1085] = {x=-0.495073, y=-27.501798, z=96.643974, rx=178.000387, ry=0.000296, rz=-0.000545, shoulder=lefty, elbow=epositive, wrist=wpositive, fatherId=frmaster[2]}
  [1086] = {x=-1.492174, y=-27.491701, z=96.642188, rx=178.000265, ry=0.000202, rz=-0.000205, shoulder=lefty, elbow=epositive, wrist=wpositive, fatherId=frmaster[2]}
  [1087] = {x=-2.497648, y=-27.483122, z=96.645521, rx=178.000127, ry=0.000072, rz=0.00014, shoulder=lefty, elbow=epositive, wrist=wpositive, fatherId=frmaster[2]}
  [1088] = {x=-3.493091, y=-27.472649, z=96.644467, rx=177.99999, ry=-0.000024, rz=0.000493, shoulder=lefty, elbow=epositive, wrist=wpositive, fatherId=frmaster[2]}
  [1089] = {x=-4.487786, y=-27.461459, z=96.648454, rx=177.999847, ry=-0.000121, rz=-0.000149, shoulder=lefty, elbow=epositive, wrist=wpositive, fatherId=frmaster[2]}
  [1090] = {x=-5.482206, y=-27.44785, z=96.642959, rx=178.000676, ry=-0.000419, rz=-0.000783, shoulder=lefty, elbow=epositive, wrist=wpositive, fatherId=frmaster[2]}
  [1091] = {x=-6.48423, y=-27.439723, z=96.638428, rx=178.000511, ry=-0.000552, rz=-0.000413, shoulder=lefty, elbow=epositive, wrist=wpositive, fatherId=frmaster[2]}
  [1092] = {x=-7.475175, y=-27.428556, z=96.648233, rx=177.99955, ry=0.000466, rz=-0.000692, shoulder=lefty, elbow=epositive, wrist=wpositive, fatherId=frmaster[2]}
  [1093] = {x=-8.475576, y=-27.420186, z=96.64446, rx=177.999368, ry=0.000329, rz=-0.00031, shoulder=lefty, elbow=epositive, wrist=wpositive, fatherId=frmaster[2]}
  [1094] = {x=-9.475849, y=-27.408282, z=96.640557, rx=178.00016, ry=-0.000002, rz=0.000078, shoulder=lefty, elbow=epositive, wrist=wpositive, fatherId=frmaster[2]}
  [1095] = {x=-10.474778, y=-27.398581, z=96.646873, rx=177.999965, ry=-0.000139, rz=0.00047, shoulder=lefty, elbow=epositive, wrist=wpositive, fatherId=frmaster[2]}
  [1096] = {x=-11.473202, y=-27.387694, z=96.643781, rx=177.999763, ry=-0.000278, rz=-0.000131, shoulder=lefty, elbow=epositive, wrist=wpositive, fatherId=frmaster[2]}
  [1097] = {x=-12.469178, y=-27.37884, z=96.650898, rx=177.998746, ry=0.00069, rz=0.00062, shoulder=lefty, elbow=epositive, wrist=wpositive, fatherId=frmaster[2]}
  [1098] = {x=-13.466236, y=-27.366639, z=96.648541, rx=177.999511, ry=0.000362, rz=0.000031, shoulder=lefty, elbow=epositive, wrist=wpositive, fatherId=frmaster[2]}
  [1099] = {x=-14.462432, y=-27.354964, z=96.641926, rx=178.000269, ry=0.000036, rz=0.000447, shoulder=lefty, elbow=epositive, wrist=wpositive, fatherId=frmaster[2]}
  [1100] = {x=-15.457681, y=-27.343902, z=96.640402, rx=178.000038, ry=-0.000105, rz=-0.000133, shoulder=lefty, elbow=epositive, wrist=wpositive, fatherId=frmaster[2]}
  [1101] = {x=-16.452211, y=-27.332268, z=96.643922, rx=177.9998, ry=-0.000247, rz=-0.000709, shoulder=lefty, elbow=epositive, wrist=wpositive, fatherId=frmaster[2]}
  [1102] = {x=-17.454111, y=-27.321812, z=96.643219, rx=178.000696, ry=0.000317, rz=0.000074, shoulder=lefty, elbow=epositive, wrist=wpositive, fatherId=frmaster[2]}
  [1103] = {x=-18.44696, y=-27.311325, z=96.638247, rx=178.000443, ry=0.000174, rz=-0.00049, shoulder=lefty, elbow=epositive, wrist=wpositive, fatherId=frmaster[2]}
  [1104] = {x=-19.448132, y=-27.302356, z=96.647723, rx=177.999189, ry=0.000168, rz=-0.000053, shoulder=lefty, elbow=epositive, wrist=wpositive, fatherId=frmaster[2]}
  [1105] = {x=-20.448782, y=-27.292696, z=96.643596, rx=177.999898, ry=-0.000187, rz=0.000391, shoulder=lefty, elbow=epositive, wrist=wpositive, fatherId=frmaster[2]}
  [1106] = {x=-21.439952, y=-27.278844, z=96.639321, rx=178.00061, ry=-0.000503, rz=-0.000158, shoulder=lefty, elbow=epositive, wrist=wpositive, fatherId=frmaster[2]}
  [1107] = {x=-22.437659, y=-27.27036, z=96.645363, rx=177.999492, ry=0.000405, rz=-0.00035, shoulder=lefty, elbow=epositive, wrist=wpositive, fatherId=frmaster[2]}
  [1108] = {x=-23.436433, y=-27.258561, z=96.641986, rx=178.000181, ry=0.000054, rz=0.000109, shoulder=lefty, elbow=epositive, wrist=wpositive, fatherId=frmaster[2]}
  [1109] = {x=-24.433773, y=-27.250404, z=96.648854, rx=177.99889, ry=0.000036, rz=-0.000431, shoulder=lefty, elbow=epositive, wrist=wpositive, fatherId=frmaster[2]}
  [1110] = {x=-25.431052, y=-27.238757, z=96.646305, rx=177.999565, ry=-0.000314, rz=0.000036, shoulder=lefty, elbow=epositive, wrist=wpositive, fatherId=frmaster[2]}
  [1111] = {x=-26.426322, y=-27.22766, z=96.648838, rx=177.999398, ry=0.000422, rz=-0.000134, shoulder=lefty, elbow=epositive, wrist=wpositive, fatherId=frmaster[2]}
  [1112] = {x=-27.422125, y=-27.216218, z=96.647125, rx=178.000058, ry=0.000076, rz=-0.000658, shoulder=lefty, elbow=epositive, wrist=wpositive, fatherId=frmaster[2]}
  [1113] = {x=-28.426074, y=-27.208488, z=96.641329, rx=177.999717, ry=-0.000147, rz=-0.000178, shoulder=lefty, elbow=epositive, wrist=wpositive, fatherId=frmaster[2]}
  [1114] = {x=-29.420847, y=-27.194401, z=96.644601, rx=178.000365, ry=-0.00049, rz=0.000306, shoulder=lefty, elbow=epositive, wrist=wpositive, fatherId=frmaster[2]}
  [1115] = {x=-30.413024, y=-27.185017, z=96.648858, rx=177.999174, ry=0.000399, rz=0.000153, shoulder=lefty, elbow=epositive, wrist=wpositive, fatherId=frmaster[2]}
  [1116] = {x=-31.415378, y=-27.17413, z=96.643812, rx=177.999799, ry=0.000021, rz=-0.000353, shoulder=lefty, elbow=epositive, wrist=wpositive, fatherId=frmaster[2]}
  [1117] = {x=-32.407452, y=-27.164034, z=96.648884, rx=177.999438, ry=-0.000167, rz=-0.000861, shoulder=lefty, elbow=epositive, wrist=wpositive, fatherId=frmaster[2]}
  [1118] = {x=-33.407268, y=-27.15328, z=96.644693, rx=178.000188, ry=0.000379, rz=0.000003, shoulder=lefty, elbow=epositive, wrist=wpositive, fatherId=frmaster[2]}
  [1119] = {x=-34.407375, y=-27.143495, z=96.645599, rx=177.999803, ry=0.000154, rz=0.000506, shoulder=lefty, elbow=epositive, wrist=wpositive, fatherId=frmaster[2]}
  [1120] = {x=-35.406925, y=-27.133242, z=96.642283, rx=178.000401, ry=-0.000217, rz=0.000013, shoulder=lefty, elbow=epositive, wrist=wpositive, fatherId=frmaster[2]}
  [1121] = {x=-36.397017, y=-27.119149, z=96.638837, rx=178.001001, ry=-0.00055, rz=-0.000475, shoulder=lefty, elbow=epositive, wrist=wpositive, fatherId=frmaster[2]}
  [1122] = {x=-37.393812, y=-27.110415, z=96.645694, rx=177.999737, ry=0.000288, rz=-0.000599, shoulder=lefty, elbow=epositive, wrist=wpositive, fatherId=frmaster[2]}
  [1123] = {x=-38.391659, y=-27.098415, z=96.643201, rx=178.000315, ry=-0.000079, rz=-0.00008, shoulder=lefty, elbow=epositive, wrist=wpositive, fatherId=frmaster[2]}
  [1124] = {x=-39.388333, y=-27.090196, z=96.641683, rx=177.999895, ry=-0.000307, rz=-0.000561, shoulder=lefty, elbow=epositive, wrist=wpositive, fatherId=frmaster[2]}
  [1125] = {x=-40.392748, y=-27.08017, z=96.649396, rx=177.999586, ry=0.000351, rz=0.000327, shoulder=lefty, elbow=epositive, wrist=wpositive, fatherId=frmaster[2]}
  [1126] = {x=-41.388564, y=-27.069406, z=96.643627, rx=178.000142, ry=-0.000012, rz=-0.000145, shoulder=lefty, elbow=epositive, wrist=wpositive, fatherId=frmaster[2]}
  [1127] = {x=-42.384051, y=-27.056523, z=96.637813, rx=178.000693, ry=-0.000374, rz=-0.000611, shoulder=lefty, elbow=epositive, wrist=wpositive, fatherId=frmaster[2]}
  [1128] = {x=-43.377355, y=-27.046197, z=96.642179, rx=178.000366, ry=0.00032, rz=-0.000712, shoulder=lefty, elbow=epositive, wrist=wpositive, fatherId=frmaster[2]}
  [1129] = {x=-44.380666, y=-27.035381, z=96.63734, rx=178.000893, ry=-0.000074, rz=-0.000174, shoulder=lefty, elbow=epositive, wrist=wpositive, fatherId=frmaster[2]}
  [1130] = {x=-45.373828, y=-27.025742, z=96.642607, rx=178.000431, ry=-0.000301, rz=-0.000638, shoulder=lefty, elbow=epositive, wrist=wpositive, fatherId=frmaster[2]}
  [1131] = {x=-46.374512, y=-27.016593, z=96.647942, rx=177.999076, ry=0.000479, rz=0.000271, shoulder=lefty, elbow=epositive, wrist=wpositive, fatherId=frmaster[2]}
  [1132] = {x=-47.366856, y=-27.004512, z=96.648977, rx=177.999592, ry=0.000125, rz=-0.000185, shoulder=lefty, elbow=epositive, wrist=wpositive, fatherId=frmaster[2]}
  [1133] = {x=-48.367522, y=-26.995992, z=96.645994, rx=177.999099, ry=-0.000144, rz=-0.000637, shoulder=lefty, elbow=epositive, wrist=wpositive, fatherId=frmaster[2]}
  [1134] = {x=-49.367042, y=-26.98281, z=96.642882, rx=178.000696, ry=0.000271, rz=0.000287, shoulder=lefty, elbow=epositive, wrist=wpositive, fatherId=frmaster[2]}
  [1135] = {x=-50.366818, y=-26.971914, z=96.644908, rx=178.000189, ry=0.000005, rz=0.000838, shoulder=lefty, elbow=epositive, wrist=wpositive, fatherId=frmaster[2]}
  [1136] = {x=-51.356599, y=-26.962304, z=96.647812, rx=177.999684, ry=-0.000226, rz=-0.00061, shoulder=lefty, elbow=epositive, wrist=wpositive, fatherId=frmaster[2]}
  [1137] = {x=-52.354155, y=-26.951843, z=96.641536, rx=178.000262, ry=0.000313, rz=0.000324, shoulder=lefty, elbow=epositive, wrist=wpositive, fatherId=frmaster[2]}
  [1138] = {x=-53.352057, y=-26.942559, z=96.649568, rx=177.99874, ry=0.000156, rz=-0.000121, shoulder=lefty, elbow=epositive, wrist=wpositive, fatherId=frmaster[2]}
  [1139] = {x=-54.349966, y=-26.929835, z=96.639101, rx=178.000193, ry=-0.000335, rz=-0.000554, shoulder=lefty, elbow=epositive, wrist=wpositive, fatherId=frmaster[2]}
  [1140] = {x=-55.345733, y=-26.919895, z=96.648011, rx=177.999751, ry=0.00032, rz=-0.00062, shoulder=lefty, elbow=epositive, wrist=wpositive, fatherId=frmaster[2]}
  [1141] = {x=-56.342288, y=-26.909156, z=96.647726, rx=177.999202, ry=0.00005, rz=-0.000054, shoulder=lefty, elbow=epositive, wrist=wpositive, fatherId=frmaster[2]}
  [1142] = {x=-57.347507, y=-26.899443, z=96.643364, rx=177.999632, ry=-0.000361, rz=0.000516, shoulder=lefty, elbow=epositive, wrist=wpositive, fatherId=frmaster[2]}
  [1143] = {x=-58.341956, y=-26.888088, z=96.64397, rx=178.000158, ry=0.000189, rz=0.000462, shoulder=lefty, elbow=epositive, wrist=wpositive, fatherId=frmaster[2]}
  [1144] = {x=-59.336884, y=-26.877874, z=96.649669, rx=177.999588, ry=-0.000079, rz=0.000029, shoulder=lefty, elbow=epositive, wrist=wpositive, fatherId=frmaster[2]}
  [1145] = {x=-60.331613, y=-26.865546, z=96.646142, rx=178.000007, ry=-0.000448, rz=-0.000394, shoulder=lefty, elbow=epositive, wrist=wpositive, fatherId=frmaster[2]}
  [1146] = {x=-61.333781, y=-26.855315, z=96.63859, rx=178.000498, ry=0.00007, rz=0.000564, shoulder=lefty, elbow=epositive, wrist=wpositive, fatherId=frmaster[2]}
  [1147] = {x=-62.327369, y=-26.843844, z=96.645201, rx=177.999907, ry=-0.000199, rz=-0.000863, shoulder=lefty, elbow=epositive, wrist=wpositive, fatherId=frmaster[2]}
  [1148] = {x=-63.328501, y=-26.83438, z=96.638603, rx=178.000381, ry=0.000323, rz=0.000098, shoulder=lefty, elbow=epositive, wrist=wpositive, fatherId=frmaster[2]}
  [1149] = {x=-64.321069, y=-26.823726, z=96.646163, rx=177.999776, ry=0.000055, rz=-0.000327, shoulder=lefty, elbow=epositive, wrist=wpositive, fatherId=frmaster[2]}
  [1150] = {x=-65.322561, y=-26.812157, z=96.644591, rx=178.000151, ry=-0.00034, rz=0.000257, shoulder=lefty, elbow=epositive, wrist=wpositive, fatherId=frmaster[2]}
  [1151] = {x=-66.322106, y=-26.804547, z=96.644041, rx=177.999603, ry=0.000275, rz=0.000218, shoulder=lefty, elbow=epositive, wrist=wpositive, fatherId=frmaster[2]}
  [1152] = {x=-67.313507, y=-26.792649, z=96.643352, rx=177.999972, ry=-0.00008, rz=-0.000196, shoulder=lefty, elbow=epositive, wrist=wpositive, fatherId=frmaster[2]}
  [1153] = {x=-66.58992, y=-27.120777, z=97.587565, rx=178.208928, ry=-0.890232, rz=-0.014201, shoulder=lefty, elbow=epositive, wrist=wpositive, fatherId=frmaster[2]}
  [1154] = {x=-66.483974, y=-27.74217, z=98.013131, rx=178.584108, ry=-1.412531, rz=-0.016752, shoulder=lefty, elbow=epositive, wrist=wpositive, fatherId=frmaster[2]}
  [1155] = {x=-65.852779, y=-27.849347, z=98.198222, rx=179.107176, ry=-1.789959, rz=-0.013253, shoulder=lefty, elbow=epositive, wrist=wpositive, fatherId=frmaster[2]}
  [1156] = {x=-65.50781, y=-28.580213, z=97.999039, rx=179.999918, ry=-1.999791, rz=0.00062, shoulder=lefty, elbow=epositive, wrist=wpositive, fatherId=frmaster[2]}
  [1157] = {x=-65.517807, y=-27.583566, z=97.994563, rx=-179.999416, ry=-2.000101, rz=-0.000767, shoulder=lefty, elbow=epositive, wrist=wpositive, fatherId=frmaster[2]}
  [1158] = {x=-65.537373, y=-26.586416, z=97.989608, rx=-179.998722, ry=-2.000403, rz=-0.000133, shoulder=lefty, elbow=epositive, wrist=wpositive, fatherId=frmaster[2]}
  [1159] = {x=-65.555558, y=-25.593676, z=97.994235, rx=-179.999923, ry=-1.999573, rz=-0.000156, shoulder=lefty, elbow=epositive, wrist=wpositive, fatherId=frmaster[2]}
  [1160] = {x=-65.575744, y=-24.595382, z=97.993273, rx=-179.999228, ry=-1.999867, rz=0.000547, shoulder=lefty, elbow=epositive, wrist=wpositive, fatherId=frmaster[2]}
  [1161] = {x=-65.586607, y=-23.600756, z=98.001848, rx=179.99945, ry=-1.999964, rz=0.000251, shoulder=lefty, elbow=epositive, wrist=wpositive, fatherId=frmaster[2]}
  [1162] = {x=-65.607339, y=-22.603, z=97.995786, rx=-179.999853, ry=-2.000241, rz=-0.000006, shoulder=lefty, elbow=epositive, wrist=wpositive, fatherId=frmaster[2]}
  [1163] = {x=-65.61888, y=-21.607999, z=97.999292, rx=179.999822, ry=-2.000425, rz=-0.000227, shoulder=lefty, elbow=epositive, wrist=wpositive, fatherId=frmaster[2]}
  [1164] = {x=-65.638891, y=-20.611228, z=97.997283, rx=179.999623, ry=-1.999661, rz=-0.000098, shoulder=lefty, elbow=epositive, wrist=wpositive, fatherId=frmaster[2]}
  [1165] = {x=-65.660263, y=-19.615604, z=97.990846, rx=-179.999678, ry=-1.999925, rz=0.000734, shoulder=lefty, elbow=epositive, wrist=wpositive, fatherId=frmaster[2]}
  [1166] = {x=-65.672709, y=-18.620098, z=97.997987, rx=180, ry=-2.000097, rz=-0.000397, shoulder=lefty, elbow=epositive, wrist=wpositive, fatherId=frmaster[2]}
  [1167] = {x=-65.685816, y=-17.622009, z=97.990602, rx=-179.999325, ry=-2.000346, rz=-0.000526, shoulder=lefty, elbow=epositive, wrist=wpositive, fatherId=frmaster[2]}
  [1168] = {x=-65.706654, y=-16.6277, z=97.996885, rx=179.999483, ry=-1.999474, rz=0.000716, shoulder=lefty, elbow=epositive, wrist=wpositive, fatherId=frmaster[2]}
  [1169] = {x=-65.720228, y=-15.630697, z=97.993712, rx=-179.999841, ry=-1.999721, rz=-0.000343, shoulder=lefty, elbow=epositive, wrist=wpositive, fatherId=frmaster[2]}
  [1170] = {x=-65.743036, y=-14.634582, z=97.990225, rx=-179.999138, ry=-1.999963, rz=0.000619, shoulder=lefty, elbow=epositive, wrist=wpositive, fatherId=frmaster[2]}
  [1171] = {x=-65.757172, y=-13.637177, z=97.995237, rx=-179.999456, ry=-2.000103, rz=-0.000407, shoulder=lefty, elbow=epositive, wrist=wpositive, fatherId=frmaster[2]}
  [1172] = {x=-65.771355, y=-12.642873, z=97.995927, rx=-179.999773, ry=-2.000238, rz=-0.000413, shoulder=lefty, elbow=epositive, wrist=wpositive, fatherId=frmaster[2]}
  [1173] = {x=-65.795044, y=-11.646523, z=97.991326, rx=-179.999067, ry=-2.000463, rz=0.000611, shoulder=lefty, elbow=epositive, wrist=wpositive, fatherId=frmaster[2]}
  [1174] = {x=-65.808962, y=-10.649054, z=97.995175, rx=-179.999285, ry=-1.999667, rz=0.000029, shoulder=lefty, elbow=epositive, wrist=wpositive, fatherId=frmaster[2]}
  [1175] = {x=-65.82402, y=-9.655133, z=97.994814, rx=-179.999599, ry=-1.999786, rz=0.000088, shoulder=lefty, elbow=epositive, wrist=wpositive, fatherId=frmaster[2]}
  [1176] = {x=-65.839633, y=-8.6583, z=97.998011, rx=-179.999914, ry=-1.999901, rz=0.000167, shoulder=lefty, elbow=epositive, wrist=wpositive, fatherId=frmaster[2]}
  [1177] = {x=-65.8556, y=-7.661804, z=97.992029, rx=-179.999231, ry=-2.000107, rz=-0.000724, shoulder=lefty, elbow=epositive, wrist=wpositive, fatherId=frmaster[2]}
  [1178] = {x=-65.871749, y=-6.665847, z=97.994594, rx=-179.999544, ry=-2.000212, rz=-0.000602, shoulder=lefty, elbow=epositive, wrist=wpositive, fatherId=frmaster[2]}
  [1179] = {x=-65.888153, y=-5.670467, z=97.996855, rx=-179.999856, ry=-2.000314, rz=-0.00046, shoulder=lefty, elbow=epositive, wrist=wpositive, fatherId=frmaster[2]}
  [1180] = {x=-65.905038, y=-4.673621, z=97.993857, rx=179.999833, ry=-2.0004, rz=-0.000322, shoulder=lefty, elbow=epositive, wrist=wpositive, fatherId=frmaster[2]}
  [1181] = {x=-65.92118, y=-3.67617, z=97.99056, rx=-179.999383, ry=-1.999677, rz=-0.00073, shoulder=lefty, elbow=epositive, wrist=wpositive, fatherId=frmaster[2]}
  [1182] = {x=-65.924201, y=-3.67615, z=107.996596, rx=-179.999579, ry=-1.999732, rz=0.000043, shoulder=lefty, elbow=epositive, wrist=wpositive, fatherId=frmaster[2]}
pointRx pdemo3 = {fatherId=frmaster[3]}
pointRx pdemo4 = {fatherId=frmaster[4]}
pointRx pdemo5 = {fatherId=frmaster[5]}
pointRx pdemo6 = {fatherId=frmaster[6]}
pointRx pdemo7 = {fatherId=frmaster[7]}
pointRx pdemo8 = {fatherId=frmaster[8]}
pointRx pdemo9 = {fatherId=frmaster[9]}
pointRx pt1 = {fatherId=world[0]}
pointRx pt2 = {x=112.095909, y=-258.119564, z=-96.596387, rx=179.943525, ry=0.071833, rz=3.231588, fatherId=world[0]}
pointRx pt3 = {fatherId=world[0]}
string sFileName[10]
  [0] = "A180"
  [1] = "A208"
  [2] = "C104"
string sFolder = "Disk://"
string smadolfrme
public tool t1 = {fatherId=flange[0], ioLink=valve1}
public tool t2[10]
  [0] = {x=44, fatherId=flange[0], ioLink=valve1}
  [1] = {fatherId=flange[0], ioLink=valve1}
  [2] = {fatherId=flange[0], ioLink=valve1}
  [3] = {fatherId=flange[0], ioLink=valve1}
  [4] = {fatherId=flange[0], ioLink=valve1}
  [5] = {x=44, fatherId=flange[0], ioLink=valve1}
  [6] = {x=44, fatherId=flange[0], ioLink=valve1}
  [7] = {x=44, fatherId=flange[0], ioLink=valve1}
  [8] = {x=44, fatherId=flange[0], ioLink=valve1}
  [9] = {x=44, fatherId=flange[0], ioLink=valve1}

--- start.pgx ---
program start()
begin
  //运行标记和暂停标记重置
  bruning=false
  bPause=false
  //创建暂停任务
  taskCreate "STOPMVE",100,SMOVE()
  //单循环停止任务
  taskCreate "sgd",100,takestop()
  //--------------------------------------------------
  //用户手动选择b0转点
  if b0==true
    for ninttool=0 to 9
      //工具值重置
      t2[ninttool].trsf={0,0,0,0,0,0}
    endFor
    //转点JOINT TO POINT程序
    call JTPdemo()
  endIf
  //

  //用户手动激活b1套用已保存的打磨坐标系
  if b1==true
    call tooolAndFrame()
  endIf
  //用户手动激活b2保存当前所有打磨坐标系
  if b2==true
    call SAVEtoolAfranme()
  endIf
  //------b3套用旧的码垛坐标系，此功能未写
  if b3==true
    call oldmaduofrme()
  endIf
  //------b4把现有的码垛坐标系保存进库，此功能未写
  if b4==true
    call saveOldframe()
  endIf
  //获取当前位置
  jchack=herej()
  //比较当前位置
  wait(jchack==jstart)
  //等待按钮状态
  wait(distart==true)
  wait(distart==false)
  //运行标记开启，暂停标记false
  bruning=true
  bPause=false
  //上电，远程模式
  enablePower()
  //检测上电
  wait(isPowered()==true)
  //开始运行码垛以及走轨迹程序
  while true
    call madol()
    waitEndMove()
  endWhile
end

--- JTPdemo.pgx ---
program JTPdemo()
  local num l_nj
begin
  //根据用户选择bA[0至9]，选择性转换单个或多个程序的joint点并使用
  //---------------------------------------------------------------------------0
  nmaster=0
  if bA[0]==true
    //加载动态库     disk://+用户输入程序名称
    call loadmaster0(sFolder+sFileName[0])
    delay(0)
    resize(nPeak0,1,1)
    l_nj=0
    //setFrame(pt1,pt2,pt3,frmaster)
    for nmaster=0 to nsize[0]-1
      pdemo0[nmaster]=jointToPoint(t2[0],frmaster[0],master:ptRoutingPath[nmaster])
      if nmaster!=0 and abs(master:ptRoutingPath[nmaster-1].j6-master:ptRoutingPath[nmaster].j6)>50
        //如果超出50，则把nmaster的数据赋值到nPeak[l_nj]
        nPeak0[l_nj]=nmaster
        //l_nj自加1
        l_nj=l_nj+1
        delay(0)
        //插入nPwak一个个数，变成可l_nj[l_nj+1]
        insert(nPeak0[l_nj])
      endIf
    endFor
    //多了一个，删除
    // delete(nPeak0[l_nj])
  endIf
  //-------------------------------------------------------------------------1
  if bA[1]==true
    nmaster=0
    call loadmaster1(sFolder+sFileName[1])
    delay(0)
    resize(nPeak1,1,1)
    l_nj=0
    for nmaster=0 to nsize[1]-1
      pdemo1[nmaster]=jointToPoint(t2[1],frmaster[1],master:ptRoutingPath[nmaster])
      if nmaster!=0 and abs(master:ptRoutingPath[nmaster-1].j6-master:ptRoutingPath[nmaster].j6)>50
        //如果超出50，则把nmaster的数据赋值到nPeak[l_nj]
        nPeak1[l_nj]=nmaster
        //l_nj自加1
        l_nj=l_nj+1
        delay(0)
        //插入nPwak一个个数，变成可l_nj[l_nj+1]
        insert(nPeak1[l_nj])
      endIf
    endFor
    //多了一个，删除
    // delete(nPeak1[l_nj])
  endIf
  //-------------------------------------------------------------------------------2
  if bA[2]==true
    nmaster=0
    call loadmaster2(sFolder+sFileName[2])
    delay(0)
    resize(nPeak2,1,1)
    l_nj=0
    //setFrame(pt1,pt2,pt3,frmaster)
    for nmaster=0 to nsize[2]-1
      pdemo2[nmaster]=jointToPoint(t2[2],frmaster[2],master:ptRoutingPath[nmaster])
      if nmaster!=0 and abs(master:ptRoutingPath[nmaster-1].j6-master:ptRoutingPath[nmaster].j6)>50
        //如果超出50，则把nmaster的数据赋值到nPeak[l_nj]
        nPeak2[l_nj]=nmaster
        //l_nj自加1
        l_nj=l_nj+1
        delay(0)
        //插入nPwak一个个数，变成可l_nj[l_nj+1]
        insert(nPeak2[l_nj])
      endIf
    endFor
    //多了一个，删除
    // delete(nPeak2[l_nj])
  endIf
  //------------------------------------------------------------------3
  if bA[3]==true
    nmaster=0
    call loadmaster3(sFolder+sFileName[3])
    delay(0)
    resize(nPeak3,1,1)
    l_nj=0
    //setFrame(pt1,pt2,pt3,frmaster)
    for nmaster=0 to nsize[3]-1
      pdemo3[nmaster]=jointToPoint(t2[3],frmaster[3],master:ptRoutingPath[nmaster])
      if nmaster!=0 and abs(master:ptRoutingPath[nmaster-1].j6-master:ptRoutingPath[nmaster].j6)>50
        //如果超出50，则把nmaster的数据赋值到nPeak[l_nj]
        nPeak3[l_nj]=nmaster
        //l_nj自加1
        l_nj=l_nj+1
        delay(0)
        //插入nPwak一个个数，变成可l_nj[l_nj+1]
        insert(nPeak3[l_nj])
      endIf
    endFor
    //多了一个，删除
    // delete(nPeak3[l_nj])
  endIf
  //---------------------------------------------------------------------------4
  if bA[4]==true
    nmaster=0
    call loadmaster4(sFolder+sFileName[4])
    delay(0)
    resize(nPeak4,1,1)
    l_nj=0
    //setFrame(pt1,pt2,pt3,frmaster)
    for nmaster=0 to nsize[4]-1
      pdemo4[nmaster]=jointToPoint(t2[4],frmaster[4],master:ptRoutingPath[nmaster])
      if nmaster!=0 and abs(master:ptRoutingPath[nmaster-1].j6-master:ptRoutingPath[nmaster].j6)>50
        //如果超出50，则把nmaster的数据赋值到nPeak[l_nj]
        nPeak4[l_nj]=nmaster
        //l_nj自加1
        l_nj=l_nj+1
        delay(0)
        //插入nPwak一个个数，变成可l_nj[l_nj+1]
        insert(nPeak4[l_nj])
      endIf
    endFor
    //多了一个，删除
    // delete(nPeak4[l_nj])
  endIf
  //-----------------------------------------------------------------------5
  if bA[5]==true
    nmaster=0
    call loadmaster5(sFolder+sFileName[5])
    delay(0)
    resize(nPeak5,1,1)
    l_nj=0
    //setFrame(pt1,pt2,pt3,frmaster)
    for nmaster=0 to nsize[5]-1
      pdemo5[nmaster]=jointToPoint(t2[5],frmaster[5],master:ptRoutingPath[nmaster])
      if nmaster!=0 and abs(master:ptRoutingPath[nmaster-1].j6-master:ptRoutingPath[nmaster].j6)>50
        //如果超出50，则把nmaster的数据赋值到nPeak[l_nj]
        nPeak5[l_nj]=nmaster
        //l_nj自加1
        l_nj=l_nj+1
        delay(0)
        //插入nPwak一个个数，变成可l_nj[l_nj+1]
        insert(nPeak5[l_nj])
      endIf
    endFor
    //多了一个，删除
    // delete(nPeak5[l_nj])
  endIf
  //-------------------------------------------------------------------6
  if bA[6]==true
    nmaster=0
    call loadmaster6(sFolder+sFileName[6])
    delay(0)
    resize(nPeak6,1,1)
    l_nj=0
    //setFrame(pt1,pt2,pt3,frmaster)
    for nmaster=0 to nsize[6]-1
      pdemo6[nmaster]=jointToPoint(t2[6],frmaster[6],master:ptRoutingPath[nmaster])
      if nmaster!=0 and abs(master:ptRoutingPath[nmaster-1].j6-master:ptRoutingPath[nmaster].j6)>50
        //如果超出50，则把nmaster的数据赋值到nPeak[l_nj]
        nPeak6[l_nj]=nmaster
        //l_nj自加1
        l_nj=l_nj+1
        delay(0)
        //插入nPwak一个个数，变成可l_nj[l_nj+1]
        insert(nPeak6[l_nj])
      endIf
    endFor
    //多了一个，删除
    //delete(nPeak6[l_nj])
  endIf
  //-------------------------------------------------------------------------------7
  if bA[7]==true
    nmaster=0
    call loadmaster7(sFolder+sFileName[7])
    delay(0)
    resize(nPeak7,1,1)
    l_nj=0
    //setFrame(pt1,pt2,pt3,frmaster)
    for nmaster=0 to nsize[7]-1
      pdemo7[nmaster]=jointToPoint(t2[7],frmaster[7],master:ptRoutingPath[nmaster])
      if nmaster!=0 and abs(master:ptRoutingPath[nmaster-1].j6-master:ptRoutingPath[nmaster].j6)>50
        //如果超出50，则把nmaster的数据赋值到nPeak[l_nj]
        nPeak7[l_nj]=nmaster
        //l_nj自加1
        l_nj=l_nj+1
        //插入nPwak一个个数，变成可l_nj[l_nj+1]
        insert(nPeak7[l_nj])
        delay(0)
      endIf
    endFor
    //多了一个，删除
    // delete(nPeak7[l_nj])
  endIf
  //----------------------------------------------------------------------------------8
  if bA[8]==true
    nmaster=0
    call loadmaster8(sFolder+sFileName[8])
    delay(0)
    resize(nPeak8,1,1)
    l_nj=0
    //setFrame(pt1,pt2,pt3,frmaster)
    for nmaster=0 to nsize[8]-1
      pdemo8[nmaster]=jointToPoint(t2[8],frmaster[8],master:ptRoutingPath[nmaster])
      if nmaster!=0 and abs(master:ptRoutingPath[nmaster-1].j6-master:ptRoutingPath[nmaster].j6)>50
        //如果超出50，则把nmaster的数据赋值到nPeak[l_nj]
        nPeak8[l_nj]=nmaster
        //l_nj自加1
        l_nj=l_nj+1
        //插入nPwak一个个数，变成可l_nj[l_nj+1]
        insert(nPeak8[l_nj])
        delay(0)
      endIf
    endFor
    //多了一个，删除
    // delete(nPeak8[l_nj])
  endIf
  //------------------------------------------------------------------------------9
  if bA[9]==true
    nmaster=0
    call loadmaster9(sFolder+sFileName[9])
    delay(0)
    resize(nPeak9,1,1)
    l_nj=0
    //setFrame(pt1,pt2,pt3,frmaster)
    for nmaster=0 to nsize[9]-1
      pdemo9[nmaster]=jointToPoint(t2[9],frmaster[9],master:ptRoutingPath[nmaster])
      if nmaster!=0 and abs(master:ptRoutingPath[nmaster-1].j6-master:ptRoutingPath[nmaster].j6)>50
        //如果超出50，则把nmaster的数据赋值到nPeak[l_nj]
        nPeak9[l_nj]=nmaster
        //l_nj自加1
        l_nj=l_nj+1
        delay(0)
        //插入nPwak一个个数，变成可l_nj[l_nj+1]
        insert(nPeak9[l_nj])
      endIf
    endFor
    //多了一个，删除
    // delete(nPeak9[l_nj])
  endIf
end

--- loadmaster0.pgx ---
program loadmaster0(string x_sMasterFile0)
begin
  if master:libLoad(x_sMasterFile0)<0
    popUpMsg("nO ok")
  endIf
  //由于mastercam生成出来的真实坐标位置是保存在tTool里的。
  frmaster[0].trsf=master:tTool.trsf
  //取个数
  nsize[0]=size(master:ptRoutingPath)
  //存个数
  resize(pdemo0,1,nsize[0])
  //保存程序
  master:libSave()
end

--- loadmaster1.pgx ---
program loadmaster1(string x_sMasterFile1 (dimensions=1))
begin
  if master:libLoad(x_sMasterFile1)<0
    popUpMsg("nO ok")
  endIf
  frmaster[1].trsf=master:tTool.trsf
  //取个数
  nsize[1]=size(master:ptRoutingPath)
  //存个数
  resize(pdemo1,1,nsize[1])
  //保存程序
  master:libSave()
end

--- loadmaster2.pgx ---
program loadmaster2(string x_sMasterFile2 (dimensions=1))
begin
  if master:libLoad(x_sMasterFile2)<0
    popUpMsg("nO ok")
  endIf
  frmaster[2].trsf=master:tTool.trsf
  //取个数
  nsize[2]=size(master:ptRoutingPath)
  //存个数
  resize(pdemo2,1,nsize[2])
  //保存程序
  master:libSave()
end

--- loadmaster3.pgx ---
program loadmaster3(string x_sMasterFile3 (dimensions=1))
begin
  if master:libLoad(x_sMasterFile3)<0
    popUpMsg("nO ok")
  endIf
  frmaster[3].trsf=master:tTool.trsf
  //取个数
  nsize[3]=size(master:ptRoutingPath)
  //存个数
  resize(pdemo3,1,nsize[3])
  //保存程序
  master:libSave()
end

--- loadmaster4.pgx ---
program loadmaster4(string x_sMasterFile4 (dimensions=1))
begin
  if master:libLoad(x_sMasterFile4)<0
    popUpMsg("nO ok")
  endIf
  frmaster[4].trsf=master:tTool.trsf
  //取个数
  nsize[4]=size(master:ptRoutingPath)
  //存个数
  resize(pdemo4,1,nsize[4])
  //保存程序
  master:libSave()
end

--- loadmaster5.pgx ---
program loadmaster5(string x_sMasterFile5 (dimensions=1))
begin
  if master:libLoad(x_sMasterFile5)<0
    popUpMsg("nO ok")
  endIf
  frmaster[5].trsf=master:tTool.trsf
  //取个数
  nsize[5]=size(master:ptRoutingPath)
  //存个数
  resize(pdemo5,1,nsize[5])
  //保存程序
  master:libSave()
end

--- loadmaster6.pgx ---
program loadmaster6(string x_sMasterFile6 (dimensions=1))
begin
  if master:libLoad(x_sMasterFile6)<0
    popUpMsg("nO ok")
  endIf
  frmaster[6].trsf=master:tTool.trsf
  //取个数
  nsize[6]=size(master:ptRoutingPath)
  //存个数
  resize(pdemo6,1,nsize[6])
  //保存程序
  master:libSave()
end

--- loadmaster7.pgx ---
program loadmaster7(string x_sMasterFile7 (dimensions=1))
begin
  if master:libLoad(x_sMasterFile7)<0
    popUpMsg("nO ok")
  endIf
  frmaster[7].trsf=master:tTool.trsf
  //取个数
  nsize[7]=size(master:ptRoutingPath)
  //存个数
  resize(pdemo7,1,nsize[7])
  //保存程序
  master:libSave()
end

--- loadmaster8.pgx ---
program loadmaster8(string x_sMasterFile8 (dimensions=1))
begin
  if master:libLoad(x_sMasterFile8)<0
    popUpMsg("nO ok")
  endIf
  frmaster[8].trsf=master:tTool.trsf
  //取个数
  nsize[8]=size(master:ptRoutingPath)
  //存个数
  resize(pdemo8,1,nsize[8])
  //保存程序
  master:libSave()
end

--- loadmaster9.pgx ---
program loadmaster9(string x_sMasterFile9 (dimensions=1))
begin
  if master:libLoad(x_sMasterFile9)<0
    popUpMsg("nO ok")
  endIf
  frmaster[9].trsf=master:tTool.trsf
  //取个数
  nsize[9]=size(master:ptRoutingPath)
  //存个数
  resize(pdemo9,1,nsize[9])
  //保存程序
  master:libSave()
end

--- madol.pgx ---
program madol()
  local num l_nj
begin
  //
  n2=0
  waitEndMove()
  //码盘for循环，3x3
  for ni=0 to 2 step 1
    for nc=0 to 2 step 1
      //抓取准备点
      movej(jready,t1,m1)
      do
        //检测吸真空状态
        if dixi==false
          //p1抓取点正上方
          movel(compose(p1,f1,{nc*180,ni*100,0,0,0,0}),t1,m1)
          //p2抓取点
          movel(compose(p2,f1,{nc*180,ni*100,0,0,0,0}),t1,m1)
          waitEndMove()
          //输出吸真空
          doxi=true
          delay(0.8)
          movel(compose(p1,f1,{nc*180,ni*100,0,0,0,0}),t1,m1)
          waitEndMove()
          //计算次数
          n2=n2+1
          waitEndMove()
        endIf
        //如果两次无料
        if n2==2
          movel(compose(p1,f1,{nc*180,ni*100,0,0,0,0}),t1,m1)
          waitEndMove()
          //暂停
          stopMove()
          //标记切换状态
          bruning=false
          bPause=true
          doxi=false
          n2=0
          waitEndMove()
          //等待启动按钮触发
          wait(distart==true)
          waitEndMove()
          //继续运行
          restartMove()
          movel(compose(p2,f1,{nc*180,ni*100,0,0,0,0}),t1,m1)
          waitEndMove()
          doxi=true
          delay(0.5)
          movel(compose(p1,f1,{nc*180,ni*100,0,0,0,0}),t1,m1)
          waitEndMove()
        endIf
      until dixi==true
      //重置吸料检测次数
      n2=0
      //准备打磨点
      movej(jbegin,t1,m1)
      waitEndMove()
      //偏移量。。输出屏幕
      nPYtest=nPY*-0.003
      gotoxy(1,1)
      put(nPYtest)
      //=========================================================
      //一整段打磨程序
      call proDEMO()
      waitEndMove()
      //------------------------------------------------------------------------------------
      waitEndMove()
      //生产工件数量+1
      nPY=nPY+1
      //npyb是触发打磨x个向下补偿一次
      nPYB=nPYB+1
      if nPYB==1
        //npyc是直接补偿
        nPYC=nPYC+1
        nPYB=0
      endIf
      //这是客户要求的阻碍开关 打磨完阻碍再jbegin点
      if ditab==true
        movej(jbegin,t1,m1)
        waitEndMove()
        //暂停
        stopMove()
        //等待这个切换开关关闭
        wait(ditab==false)
        restartMove()
      endIf
      //打磨结束连接点
      movej(jend,t1,m1)
      waitEndMove()
      //卸料点
      movej(jXieLiao,t1,m1)
      waitEndMove()
      //吸真空关闭，吹气开启卸料
      doxi=false
      dochui=true
      waitEndMove()
      delay(0.2)
      waitEndMove()
      wait(dixi==false)
      dochui=false
      //
      movej(jXieLiao,t1,m1)
      delay(0.5)
      //客户自己添加的一个卸料感应程序
      if diganying==true
        //单循环阻碍的一个条件
        bstop=true
      endIf
      //回到原点
      movej(jstart,t1,m1)
      waitEndMove()
      //当做了2000个时，补偿置0，更换砂带
      if nPY==2000
        stopMove()
        gotoxy(5,5)
        popUpMsg("1000次补偿完成，请更换砂带")
        nPYC=0
        nPY=0
        nPYtest=0
        //等待更换砂带后触发条件
        wait(distart==true)
        restartMove()
      endIf
      //这里bstop阻碍整个程序的运行，也就是单循环停止
      wait(bstop==false)
    endFor
  endFor
  waitEndMove()
end

--- oldmaduofrme.pgx ---
program oldmaduofrme()
begin
  f1.trsf=lib:fr1.trsf
  t1.trsf=lib:t1.trsf
end

--- proDEMO.pgx ---
program proDEMO()
  local num l_nj
begin
  //这是程序运行的选择，根据用户选择的bA[0至9]状态运行单个或多个程序
  //----------------------------------------------------------------0
  if bA[0]==true
    //movej(jA[0],t2[0],m1)
    movej(pdemo0[0],t2[0],m1)
    waitEndMove()
    ndemo=0
    //重置l_nj
    l_nj=0
    for ndemo=0 to nsize[0]-1
      //当ndemo和nPeak相等时
      if ndemo==nPeak0[l_nj] and nPeak0[l_nj]!=0
        //速度加快
        movej(compose(pdemo0[ndemo],frmaster[0],{0,0,nPYC*-0.002,0,0,0}),t2[0],mFast)
        //自加1，等待下一个点加速
        l_nj=l_nj+1
        delay(0)
        //否则使用普通速度
      else
        movej(compose(pdemo0[ndemo],frmaster[0],{0,0,nPYC*-0.002,0,0,0}),t2[0],mSuDu[1])
      endIf
    endFor
    //movej(jA[1],t2[0],m1)
    movej(pdemo0[nsize[0]-1],t2[0],m1)
    waitEndMove()
  endIf
  //---------------------------------------------------------------------------------1
  if bA[1]==true
    //movej(jA[2],t2[1],m1)
    movej(pdemo1[0],t2[1],m1)
    waitEndMove()
    ndemo=0
    //重置l_nj
    l_nj=0
    for ndemo=0 to nsize[1]-1
      //当ndemo和nPeak相等时
      if ndemo==nPeak1[l_nj] and nPeak1[l_nj]!=0
        //速度加快
        movej(compose(pdemo1[ndemo],frmaster[1],{0,0,nPYC*-0.002,0,0,0}),t2[1],mFast)
        //自加1，等待下一个点加速
        l_nj=l_nj+1
        delay(0)
        //否则使用普通速度
      else
        movej(compose(pdemo1[ndemo],frmaster[1],{0,0,nPYC*-0.002,0,0,0}),t2[1],mSuDu[1])
      endIf
    endFor
    //movej(jA[3],t2[1],m1)
    movej(pdemo1[nsize[1]-1],t2[1],m1)
    waitEndMove()
  endIf
  //----------------------------------------------------------------------------------------2
  if bA[2]==true
    //movej(jA[4],t2[2],m1)
    movej(pdemo2[0],t2[2],m1)
    waitEndMove()
    ndemo=0
    //重置l_nj
    l_nj=0
    for ndemo=0 to nsize[2]-1
      //当ndemo和nPeak相等时
      if ndemo==nPeak2[l_nj] and nPeak2[l_nj]!=0
        //速度加快
        movej(compose(pdemo2[ndemo],frmaster[2],{0,0,nPYC*-0.002,0,0,0}),t2[2],mFast)
        //自加1，等待下一个点加速
        l_nj=l_nj+1
        delay(0)
        //否则使用普通速度
      else
        movej(compose(pdemo2[ndemo],frmaster[2],{0,0,nPYC*-0.002,0,0,0}),t2[2],mSuDu[1])
      endIf
    endFor
    //movej(jA[5],t2[2],m1)
    movej(pdemo2[nsize[2]-1],t2[2],m1)
    waitEndMove()
  endIf
  //------------------------------------------------------------------------------------3
  if bA[3]==true
    //movej(jA[6],t2[3],m1)
    movej(pdemo3[0],t2[3],m1)
    waitEndMove()
    ndemo=0
    //重置l_nj
    l_nj=0
    for ndemo=0 to nsize[3]-1
      //当ndemo和nPeak相等时
      if ndemo==nPeak3[l_nj] and nPeak3[l_nj]!=0
        //速度加快
        movej(compose(pdemo3[ndemo],frmaster[3],{0,0,nPYC*-0.002,0,0,0}),t2[3],mFast)
        //自加1，等待下一个点加速
        l_nj=l_nj+1
        delay(0)
        //否则使用普通速度
      else
        movej(compose(pdemo3[ndemo],frmaster[3],{0,0,nPYC*-0.002,0,0,0}),t2[3],mSuDu[1])
      endIf
    endFor
    //movej(jA[7],t2[3],m1)
    movej(pdemo3[nsize[3]-1],t2[3],m1)
    waitEndMove()
  endIf
  //-----------------------------------------------------------------------------------4
  if bA[4]==true
    // movej(jA[8],t2[4],m1)
    movej(pdemo4[0],t2[4],m1)
    waitEndMove()
    ndemo=0
    //重置l_nj
    l_nj=0
    for ndemo=0 to nsize[4]-1
      //当ndemo和nPeak相等时
      if ndemo==nPeak4[l_nj] and nPeak4[l_nj]!=0
        //速度加快
        movej(compose(pdemo4[ndemo],frmaster[4],{0,0,nPYC*-0.002,0,0,0}),t2[4],mFast)
        //自加1，等待下一个点加速
        l_nj=l_nj+1
        delay(0)
        //否则使用普通速度
      else
        movej(compose(pdemo4[ndemo],frmaster[4],{0,0,nPYC*-0.002,0,0,0}),t2[4],mSuDu[1])
      endIf
    endFor
    //movej(jA[9],t2[4],m1)
    movej(pdemo4[nsize[4]-1],t2[4],m1)
    waitEndMove()
  endIf
  //-------------------------------------------------------------------------------------5
  if bA[5]==true
    //movej(jA[10],t2[5],m1)
    movej(pdemo5[0],t2[5],m1)
    waitEndMove()
    ndemo=0
    //重置l_nj
    l_nj=0
    for ndemo=0 to nsize[5]-1
      //当ndemo和nPeak相等时
      if ndemo==nPeak5[l_nj] and nPeak5[l_nj]!=0
        //速度加快
        movej(compose(pdemo5[ndemo],frmaster[5],{0,0,nPYC*-0.002,0,0,0}),t2[5],mFast)
        //自加1，等待下一个点加速
        l_nj=l_nj+1
        delay(0)
        //否则使用普通速度
      else
        movej(compose(pdemo5[ndemo],frmaster[5],{0,0,nPYC*-0.002,0,0,0}),t2[5],mSuDu[1])
      endIf
    endFor
    //movej(jA[11],t2[5],m1)
    movej(pdemo5[nsize[5]-1],t2[5],m1)
    waitEndMove()
  endIf
  //---------------------------------------------------------------------------------6
  if bA[6]==true
    //movej(jA[12],t2[6],m1)
    movej(pdemo6[0],t2[6],m1)
    waitEndMove()
    ndemo=0
    //重置l_nj
    l_nj=0
    for ndemo=0 to nsize[6]-1
      //当ndemo和nPeak相等时
      if ndemo==nPeak6[l_nj] and nPeak6[l_nj]!=0
        //速度加快
        movej(compose(pdemo6[ndemo],frmaster[6],{0,0,nPYC*-0.002,0,0,0}),t2[6],mFast)
        //自加1，等待下一个点加速
        l_nj=l_nj+1
        delay(0)
        //否则使用普通速度
      else
        movej(compose(pdemo6[ndemo],frmaster[6],{0,0,nPYC*-0.002,0,0,0}),t2[6],mSuDu[1])
      endIf
    endFor
    //movej(jA[13],t2[6],m1)
    movej(pdemo6[nsize[6]-1],t2[6],m1)
    waitEndMove()
  endIf
  //-----------------------------------------------------------------------------------7
  if bA[7]==true
    //movej(jA[14],t2[7],m1)
    movej(pdemo7[0],t2[7],m1)
    waitEndMove()
    ndemo=0
    //重置l_nj
    l_nj=0
    for ndemo=0 to nsize[7]-1
      //当ndemo和nPeak相等时
      if ndemo==nPeak7[l_nj] and nPeak7[l_nj]!=0
        //速度加快
        movej(compose(pdemo7[ndemo],frmaster[7],{0,0,nPYC*-0.002,0,0,0}),t2[7],mFast)
        //自加1，等待下一个点加速
        l_nj=l_nj+1
        delay(0)
        //否则使用普通速度
      else
        movej(compose(pdemo7[ndemo],frmaster[7],{0,0,nPYC*-0.002,0,0,0}),t2[7],mSuDu[1])
      endIf
    endFor
    //movej(jA[15],t2[7],m1)
    movej(pdemo7[nsize[7]-1],t2[7],m1)
    waitEndMove()
  endIf
  //--------------------------------------------------------------------------8
  if bA[8]==true
    //movej(jA[16],t2[8],m1)
    movej(pdemo8[0],t2[8],m1)
    waitEndMove()
    ndemo=0
    //重置l_nj
    l_nj=0
    for ndemo=0 to nsize[8]-1
      //当ndemo和nPeak相等时
      if ndemo==nPeak8[l_nj] and nPeak8[l_nj]!=0
        //速度加快
        movej(compose(pdemo8[ndemo],frmaster[8],{0,0,nPYC*-0.002,0,0,0}),t2[8],mFast)
        //自加1，等待下一个点加速
        l_nj=l_nj+1
        delay(0)
        //否则使用普通速度
      else
        movej(compose(pdemo8[ndemo],frmaster[8],{0,0,nPYC*-0.002,0,0,0}),t2[8],mSuDu[1])
      endIf
    endFor
    //movej(jA[17],t2[8],m1)
    movej(pdemo8[nsize[8]-1],t2[8],m1)
    waitEndMove()
  endIf
  //-----------------------------------------------------------------------------------------9
  if bA[9]==true
    // movej(jA[18],t2[9],m1)
    movej(pdemo9[0],t2[9],m1)
    waitEndMove()
    ndemo=0
    //重置l_nj
    l_nj=0
    for ndemo=0 to nsize[9]-1
      //当ndemo和nPeak相等时
      if ndemo==nPeak9[l_nj] and nPeak9[l_nj]!=0
        //速度加快
        movej(compose(pdemo9[ndemo],frmaster[9],{0,0,nPYC*-0.002,0,0,0}),t2[9],mFast)
        //自加1，等待下一个点加速
        l_nj=l_nj+1
        delay(0)
        //否则使用普通速度
      else
        movej(compose(pdemo9[ndemo],frmaster[9],{0,0,nPYC*-0.002,0,0,0}),t2[9],mSuDu[1])
      endIf
    endFor
    // movej(jA[19],t2[9],m1)
    movej(pdemo9[nsize[9]-1],t2[9],m1)
    waitEndMove()
  endIf
end

--- saveOldframe.pgx ---
program saveOldframe()
begin
  lib:fr1.trsf=f1.trsf
  lib:t1.trsf=t1.trsf
end

--- SAVEtoolAfranme.pgx ---
program SAVEtoolAfranme()
begin
  for nframe=0 to 9
    lib:frmaster[nframe].trsf=frmaster[nframeSave[nframe]].trsf
  endFor
  for ntool=0 to 9
    lib:t2[ntool].trsf=t2[ntoolSave[ntool]].trsf
  endFor
end

--- SMOVE.pgx ---
program SMOVE()
begin
  //
  while true
    if bruning==true and distart==true
      stopMove()
      bPause=true
      bruning=false
      wait(distart==false)
    endIf
    if bPause and distart==true
      restartMove()
      bruning=true
      bPause=false
      wait(distart==false)
    endIf
    delay(0)
  endWhile
end

--- takestop.pgx ---
program takestop()
begin
  //
  while true
    if distop==true
      bstop=true
    endIf
    if distart==true
      bstop=false
    endIf
    delay(0)
  endWhile
end

--- tooolAndFrame.pgx ---
program tooolAndFrame()
begin
  for nframe=0 to 9
    frmaster[nframe].trsf=lib:frmaster[nframeSave[nframe]].trsf
    delay(0)
  endFor
  for ntool=0 to 9
    t2[ntool].trsf=lib:t2[ntoolSave[ntool]].trsf
    delay(0)
  endFor
end
